(* CODESYS project FCC-Demo
   Author: Luke
   Company: Electra
   CompiledLibraryCompatibilityVersion: CODESYS V3.5 SP13
   Description: Reduced Brusa Temps for fan
      ePTO set to activate with reverse
      Cooling Fan reinstated
      Additional compressor run signals
      Gear change adjustment
      Comp temp Error SP raised
      Auto regen on overspeed >56@5s
      OR t AND for Traction Off Keypad Combo
   Title: e-Compact
   Version: 3.0.6

Project tree, tasks and I/O mapping:
  application Application
    libraries: SAE J1939, 3.0.9.1 (Epec Oy); Event Log, 3.3.0.0 (Epec Oy); CmpApp, * (System); CmpErrors, * (System); AD Conversion, 3.0.2.5 (Epec Oy); Analog Input, 3.0.0.5 (Epec Oy); CANopen, 3.5.4.3 (Epec Oy); CANopen 302, 3.0.2.2 (Epec Oy); CANopenCSDO, 3.1.3.1 (Epec Oy); CANopen OD Save, 3.3.3.8 (Epec Oy); Digital Output Diagnostic, 3.0.2.1 (Epec Oy); Event Log GUI, 3.0.1.9 (Epec Oy); Event Log Transfer, 3.0.4.4 (Epec Oy); RAM File System, 3.2.0.3 (Epec Oy); J1939 To Event Translator, 3.0.1.0 (Epec Oy); Filters, 3.0.1.4 (Epec Oy); Network Manager, 3.2.4.8 (Epec Oy); 5000types, 3.5.7.2 (Epec Oy); Joystick Calibration And Diagnostic, 3.2.0.6 (Epec Oy); Proportional Valve Control, 3.0.3.0 (Epec Oy); Ramp, 3.0.1.0 (Epec Oy); Sensor Calibration And Diagnostic, 3.0.1.6 (Epec Oy); DataTransfer, 3.0.2.0 (Epec Oy); CANVXD API, 4.0.0.1 (Epec Oy); Parameter Handler, 1.0.0.10 (Epec Oy); CANL2 CANVXD, 4.0.0.2 (Epec Oy); CANVXD API, 4.0.0.1 (Epec Oy); Util, * (System); BASIC, 3.3.4.0 (OSCAT)
    task PLC_PRG_TASK (cyclic, interval 10 ms, priority 1) calls PLC_PRG
    global variables ChangeLog
    CodeTemplate/
      Constants/
        global variables Code_Template_constants
      Enums/
        data type InitCanProtocolStates
      Globals/
        CANopen_CAN1/
          global variables G_CAN1_VAR
          global variables G_CANopen_CAN1
          global variables G_CANopen_CAN1_VAR
        CANopen_CAN2/
          global variables G_CAN2_VAR
          global variables G_CANopen_CAN2
          global variables G_CANopen_CAN2_VAR
        CANopen_CAN3/
          global variables G_CAN3_VAR
          global variables G_CANopen_CAN3
          global variables G_CANopen_CAN3_VAR
        CANopen_CAN4/
          global variables G_CAN4_VAR
          global variables G_CANopen_CAN4
          global variables G_CANopen_CAN4_VAR
        global variables Code_Template_globals
        global variables ERRORS
        global variables G_Common
        global variables G_SystemInfo
        global variables IO
        global variables IO_CONFIG
        global variables IO_INTERNAL
        global variables IO_RAW
        global variables J1939Globals
        global variables OD1_VAR
        global variables OD2_VAR
        global variables OD3_VAR
        global variables OD4_VAR
        global variables Slave_Configurations
        global variables SYSTEM
      POUs/
        program PLC_PRG [SFC]: Application_Action, Bus_Action, Diag_Action, EPEC_In_Action, Epec_Out_Action, Init_Action, Init_Bus_Action, Init_Entry_Action, Init_Events_Action, Init_Exit_Action, Init_Flash_Action, Init_IO_Action, Init_Protocols_Can1_Action, Init_Protocols_Can2_Action, Init_Protocols_Can3_Action, Init_Protocols_Can4_Action, IOFilter_Action, IOHandleOutputs_Action, Main_Application_Action, Other_Action, Other_EpecOut_Action
      Structs/
        CANopen/
          data type IdentityObject
        J1939/
          data type J1939_CAN1
          data type J1939_CAN1_IN
          data type J1939_CAN1_IN_BodyCont
          data type J1939_CAN1_IN_CCVS
          data type J1939_CAN1_IN_Engine
          data type J1939_CAN4
          data type J1939_CAN4_IN_ABS1
          data type J1939_CAN4_IN
          data type J1939_CAN4_IN_Tacho
    UserCode/
      BELDCDC/
        program BELDCDC_Control_1 [ST]
        program BELDCDC_Rx_1 [ST]
        program BELDCDC_RxConversion_1 [ST]
        program BELDCDC_Tx_1 [ST]
        program BELDCDC_TxConversion_1 [ST]
      BELDCDC/
        program BELDCDC_RxConversion [ST]
        program BELDCDC_Tx [ST]
        program BELDCDC_Control [ST]
        program BELDCDC_Rx [ST]
        program BELDCDC_TxConversion [ST]
        global variables BELDCDC_VAR
      BMS/
        global variables BMS_VAR
        program BMSData [ST]
        CATL/
          program CATLBMS_RxConversion [ST]
          program CATLBMS1_Rx [ST]
          global variables CATLBMS_VAR
        OrionBMS/
          program OrionBMS2_RxConversion [ST]
          global variables OrionBMS2_VAR
          program OrionBMS_Tx [ST]
          program Orion_Control [ST]
          program OrionBMS1_Rx [ST]
          program OrionBMS1_RxConversion [ST]
          global variables OrionBMS1_VAR
          program OrionBMS2_Rx [ST]
      BMS/
        global variables BMS_VAR_1
        program BMSData_1 [ST]
        CATL/
          program CATLBMS1_Rx_1 [ST]
          program CATLBMS_RxConversion_1 [ST]
          global variables CATLBMS_VAR_1
        OrionBMS/
          program Orion_Control_1 [ST]
          program OrionBMS1_Rx_1 [ST]
          program OrionBMS1_RxConversion_1 [ST]
          global variables OrionBMS1_VAR_1
          program OrionBMS2_Rx_1 [ST]
          program OrionBMS2_RxConversion_1 [ST]
          global variables OrionBMS2_VAR_1
          program OrionBMS_Tx_1 [ST]
      Brusa/
        Brusa1_Comms/
          program Brusa1_Rx_1 [ST]
          program Brusa1_RxConversion_1 [ST]
          program Brusa1_Tx_1 [ST]
          program Brusa1_TxConversion_1 [ST]
        Brusa2_Comms/
          program Brusa2_Rx_1 [ST]
          program Brusa2_RxConversion_1 [ST]
          program Brusa2_Tx_1 [ST]
          program Brusa2_TxConversion_1 [ST]
        program Brusa_1 [ST]: FreeContactor
        function block BrusaControl_1 [ST]: OkToCharge, OkToReset
      Brusa/
        Brusa1_Comms/
          program Brusa1_Rx [ST]
          program Brusa1_RxConversion [ST]
          program Brusa1_Tx [ST]
          program Brusa1_TxConversion [ST]
        Brusa2_Comms/
          program Brusa2_Rx [ST]
          program Brusa2_RxConversion [ST]
          program Brusa2_Tx [ST]
          program Brusa2_TxConversion [ST]
        program Brusa [ST]: FreeContactor
        function block BrusaControl [ST]: OkToCharge, OkToReset
      CAN1/
        program CAN1_RxConversion [ST]
        program CAN1_Rx [ST]
        program CAN1_TCMs_Tx [ST]
        program CAN1_Tx [ST]
        program CAN1_TxConversion [ST]
        global variables CAN1_VAR
        program KB_Tx [ST]
      CAN1/
        program CAN1_Rx_1 [ST]
        program CAN1_RxConversion_1 [ST]
        program CAN1_TCMs_Tx_1 [ST]
        program CAN1_Tx_1 [ST]
        program CAN1_TxConversion_1 [ST]
        global variables CAN1_VAR_1
        program KB_Tx_1 [ST]
      CAN3/
        program CAN3_Rx_1 [ST]
        program CAN3_RxConversion_1 [ST]
        program CAN3_Tx_1 [ST]
        global variables CAN3_VAR_1
      CAN3/
        program CAN3_RxConversion [ST]
        program CAN3_Rx [ST]
        program CAN3_Tx [ST]
        global variables CAN3_VAR
      CAN4/
        program CAN4_Rx [ST]
        program CAN4_Tx [ST]
        global variables CAN4_VAR
        global variables HMI_VAR
        program CAN4_TxConversion [ST]
        Data to or For HMI/
          program MCU_to_HMI [ST]
          program Sevcon_to_HMI [ST]
          program BMS_to_HMI [ST]
          program BRUSA_to_HMI [ST]
          program DCDC_to_HMI [ST]
          program VMU_to_HMI [ST]
        Heater/
          program Heater_Control [ST]
          global variables Heater_VAR
          program Heater_Rx [ST]
          program Heater_Tx [ST]
        program HMI_Rx [ST]
      CAN4/
        program CAN4_Rx_1 [ST]
        program CAN4_Tx_1 [ST]
        program CAN4_TxConversion_1 [ST]
        global variables CAN4_VAR_1
      CAN Function Blocks/
        CAN1/
          function block Receive_CAN1_EXD [ST]
          function block Callback_Receive_CAN1 [ST]: Receive
          function block Receive_CAN1_EXD_28bit [ST]
          function block Receive_CAN1_STD [ST]
        CAN3/
          function block Receive_CAN3_EXD_28bit [ST]
          function block Receive_CAN3_EXD [ST]
          function block Callback_Receive_CAN3 [ST]: Receive
          function block Receive_CAN3_STD [ST]
        data type t_CANReceive
        CAN2/
          function block Callback_Receive_CAN2 [ST]: Receive
          function block Receive_CAN2_EXD [ST]
          function block Receive_CAN2_STD [ST]
        CAN4/
          function block Receive_CAN4_EXD [ST]
          function block Callback_Receive_CAN4 [ST]: Receive
          function block Receive_CAN4_STD [ST]
      CAN Function Blocks/
        CAN1/
          function block Callback_Receive_CAN1_1 [ST]: Receive
          function block Receive_CAN1_EXD_1 [ST]
          function block Receive_CAN1_EXD_28bit_1 [ST]
          function block Receive_CAN1_STD_1 [ST]
        CAN2/
          function block Callback_Receive_CAN2_1 [ST]: Receive
          function block Receive_CAN2_EXD_1 [ST]
          function block Receive_CAN2_STD_1 [ST]
        CAN3/
          function block Callback_Receive_CAN3_1 [ST]: Receive
          function block Receive_CAN3_EXD_1 [ST]
          function block Receive_CAN3_EXD_28bit_1 [ST]
          function block Receive_CAN3_STD_1 [ST]
        CAN4/
          function block Callback_Receive_CAN4_1 [ST]: Receive
          function block Receive_CAN4_EXD_1 [ST]
          function block Receive_CAN4_STD_1 [ST]
        data type t_CANReceive_1
      CodeTemplateHandlers/
      Contactor Control/
        program ContactorControl_1 [ST]
      Contactor Control/
        program ContactorControl [ST]
      Cooling Fan/
        program Cooling_Fan [FBD]
      Cooling Fan/
        program Fan_Cooling [ST]
      Cruise Control/
        program CruiseControl [ST]
      DataTypes/
        data type tUpdate_1
      DataTypes/
        data type tUpdate
      ePTO/
        program EPTO_Rx [ST]
        global variables ePTO_VAR
        program ePTO_Control [ST]
        program EPTO_Tx [ST]
      ePTO/
        program ePTO_Control_1 [ST]
        program EPTO_Rx_1 [ST]
        program EPTO_Tx_1 [ST]
        global variables ePTO_VAR_1
      Fault Handler/
        program FaultDetection_1 [ST]
      Fault Handler/
        global variables Fault_VAR
        program FaultDetection [ST]
      Functions/
        function Update [ST]
      Functions/
        function Update_1 [ST]
      Heater/
        program Heater_Control_1 [ST]
        program Heater_Rx_1 [ST]
        program Heater_Tx_1 [ST]
      HMI/
        Data to or For HMI/
          program BMS_to_HMI_1 [ST]
          program BRUSA_to_HMI_1 [ST]
          program DCDC_to_HMI_1 [ST]
          program MCU_to_HMI_1 [ST]
          program Sevcon_to_HMI_1 [ST]
          program VMU_to_HMI_1 [ST]
        program HMI_Rx_1 [ST]
      Main Program/
        program Chassis_Parameters [ST]
        program ComponentSelection [ST]
        program Main [ST]: IO_Reconfiguration
        global variables PersistentVars
        program System_StateSpace [ST]
        function GetAppInfo [ST]
        global variables Main_VAR
        program MainInit [ST]
        program Project_Infomation [FBD]
        program RealTimeClock [FBD]
      MCU/
        program Dennis_Regen [FBD]
        program Driveability [ST]
        function f_DistanceCalc [ST]
        function f_SpeedCalc [ST]
        program MCU_Control [ST]
        program MCU_Rx [ST]
        program GearSelection [ST]
        program MCU_RxConversion [ST]
        program MCU_Tx [ST]
        program MCU_TxConversion [ST]
        global variables MCU_VAR
      MCU/
        program Dennis_Regen_1 [FBD]
        program Driveability_1 [ST]
        function f_DistanceCalc_1 [ST]
        function f_SpeedCalc_1 [ST]
        program GearSelection_1 [ST]
        program MCU_Control_1 [ST]
        program MCU_Rx_1 [ST]
        program MCU_RxConversion_1 [ST]
        program MCU_Tx_1 [ST]
        program MCU_TxConversion_1 [ST]
        global variables MCU_VAR_1
      Sevcon_Compressor/
        program Sevcon2_Rx [ST]
        program Sevcon2_RxConversion [ST]
        program Sevcon2_TxConversion [ST]
        global variables Sevcon2_VAR
        program Sevcon2_Control [ST]
        program Sevcon2_Tx [ST]
      Sevcon_Compressor/
        program Sevcon2_Control_1 [ST]
        program Sevcon2_Rx_1 [ST]
        program Sevcon2_RxConversion_1 [ST]
        program Sevcon2_Tx_1 [ST]
        program Sevcon2_TxConversion_1 [ST]
        global variables Sevcon2_VAR_1
      Sevcon ePTO/
        program Sevcon_ePTO_Control [ST]
        program Sevcon_ePTO_Rx [ST]
        program Sevcon_ePTO_RxConversion [ST]
        program Sevcon_ePTO_Tx [ST]
        program Sevcon_ePTO_TxConversion [ST]
        global variables Sevcon_ePTO_VAR
      Sevcon_PSP/
        program Sevcon_Steer_Control [ST]
        program Sevcon_Steer_Rx [ST]
        program Sevcon_Steer_RxConversion [ST]
        program Sevcon_Steer_Tx [ST]
        program Sevcon_Steer_TxConversion [ST]
        global variables Sevcon_Steer_VAR
      Sevcon_PSP/
        program Sevcon_Steer_Control_1 [ST]
        program Sevcon_Steer_Rx_1 [ST]
        program Sevcon_Steer_RxConversion_1 [ST]
        program Sevcon_Steer_Tx_1 [ST]
        program Sevcon_Steer_TxConversion_1 [ST]
        global variables Sevcon_Steer_VAR_1
      UserMramUsage_1/
        data type UserMRAMStructure_1
        global variables UserMramVariables_1
      UserMramUsage/
        data type UserMRAMStructure
        global variables UserMramVariables
  function GetLibVersion [ST]
  function GetLibVersionNumber [ST]
  function IsLibReleased [ST]
  function GetBooleanProperty [ST]
  function GetCompany [ST]
  function GetNumberProperty [ST]
  function GetTextProperty2 [ST]
  function GetTextProperty [ST]
  function GetTitle [ST]
  function GetVersion [ST]
  function GetVersionProperty [ST]
*)

// Application/CodeTemplate/Enums/InitCanProtocolStates
TYPE InitCanProtocolStates :
(
	INIT_CANOPEN_PROTOCOLS := 1,
	INIT_CANOPEN_OD := 2,
	INIT_CANOPEN_PDO := 3,
	INIT_CANOPEN_OD_SAVE := 4,
	INIT_J1939 := 5,
	INIT_PROTOCOLS_DONE := 6
);
END_TYPE

// Application/UserCode/CAN Function Blocks/t_CANReceive
TYPE t_CANReceive EXTENDS EPEC_CANL2.EPEC_CANVXD.Msg:
STRUCT
	q_NewDataRxed	:	BOOL;
END_STRUCT
END_TYPE

// Application/UserCode/CAN Function Blocks/t_CANReceive_1
TYPE t_CANReceive_1 EXTENDS EPEC_CANL2.EPEC_CANVXD.Msg:
STRUCT
	q_NewDataRxed	:	BOOL;
END_STRUCT
END_TYPE

// Application/UserCode/DataTypes/tUpdate_1
(*================================================================================================*)
(*   Screen Update Structure                                                                      *)
(*================================================================================================*)
 TYPE tUpdate_1 :
 STRUCT
  Step	        :BYTE  := 0;   // Current State
  Next	        :BYTE  := 0;   // Requested Next State 
  Last	        :BYTE  := 0;   // Last Active State
  Force	        :BYTE  := 255; // Forced Next State	
  Tmr		    :WORD  := 0;   // Time In State
  Seq		    :DWORD := 0;   // Last 4 States 

 END_STRUCT
 END_TYPE

// Application/UserCode/UserMramUsage_1/UserMRAMStructure_1
TYPE UserMRAMStructure_1 :
STRUCT
   (* Header part *)
    UserMRAMdataValid:BOOL := FALSE;	(* 	Set TRUE if data pointer is initialised correctly else set FALSE*) 
    UserMRAMinitError:INT := 0; 		(* 	Possible errors 
                    						0 = SUCCESS, 
											1 = Structure size is too big to fit in MRAM, 
											2 = Tag not AA55AA55h *)                                                         
    UserMRAMTag:DWORD:=16#AA55AA55; 	(* Tag value must always be AA55AA55h *)

	(* 	User part. Forward from here user can add own variables which are stored in MRAM.
    	NOTE!!! You can add structure members until structure size is bigger than reserved size.
        In of error in size of the MRAM pointer from system pointer G_pUserMramStructure is set to point default instance
        G_UserMramStructureDefault and dataValid is set FALSE.

        NOTE!!! It is allowed to add pointers to end of the structure but not in the between 
        already added structure members.*)

		
		
END_STRUCT
END_TYPE

// Application/UserCode/UserMramUsage/UserMRAMStructure
TYPE UserMRAMStructure :
STRUCT
   (* Header part *)
    UserMRAMdataValid:BOOL := FALSE;	(* 	Set TRUE if data pointer is initialised correctly else set FALSE*) 
    UserMRAMinitError:INT := 0; 		(* 	Possible errors 
                    						0 = SUCCESS, 
											1 = Structure size is too big to fit in MRAM, 
											2 = Tag not AA55AA55h *)                                                         
    UserMRAMTag:DWORD:=16#AA55AA55; 	(* Tag value must always be AA55AA55h *)

	(* 	User part. Forward from here user can add own variables which are stored in MRAM.
    	NOTE!!! You can add structure members until structure size is bigger than reserved size.
        In of error in size of the MRAM pointer from system pointer G_pUserMramStructure is set to point default instance
        G_UserMramStructureDefault and dataValid is set FALSE.

        NOTE!!! It is allowed to add pointers to end of the structure but not in the between 
        already added structure members.*)

		
		
END_STRUCT
END_TYPE

// Application/CodeTemplate/Structs/CANopen/IdentityObject
TYPE IdentityObject :
STRUCT
	///Vendor ID
	VendorId: DWORD := 0;
	///Product code
	ProductCode: DWORD := 0;
	///Revision number
	Revision: DWORD := 0;
	///Serial number for control unit
	SerialNumber: DWORD := 0;
END_STRUCT
END_TYPE

// Application/CodeTemplate/Structs/J1939/J1939_CAN1
TYPE J1939_CAN1 :
STRUCT
	In: J1939_CAN1_IN;
END_STRUCT
END_TYPE

// Application/CodeTemplate/Structs/J1939/J1939_CAN1_IN
TYPE J1939_CAN1_IN :
STRUCT
	BodyCont: J1939_CAN1_IN_BodyCont;
	Engine: J1939_CAN1_IN_Engine;
	CCVS: J1939_CAN1_IN_CCVS;
	PGNs: ARRAY[1..3] OF J1939_pPGN;
END_STRUCT
END_TYPE

// Application/CodeTemplate/Structs/J1939/J1939_CAN1_IN_BodyCont
TYPE J1939_CAN1_IN_BodyCont :
STRUCT
	AIR1_PneumaticSupplyPress: BYTE;
	AIR1_ParkingAnd_OrTrailerAirPress: BYTE;
	AIR1_ServiceBrakeAirPressCircuit1: BYTE;
	AIR1_ServiceBrakeAirPressCircuit2: BYTE;
	AIR1_AuxEquipmentSupplyPress: BYTE;
	AIR1_AirSuspensionSupplyPress: BYTE;
	AIR1_AirCompressorStatus: BYTE;
	PGN_AIR1_SPNs: ARRAY[1..7] OF J1939_SPN;
	PGN_AIR1: J1939_PGN;
END_STRUCT
END_TYPE

// Application/CodeTemplate/Structs/J1939/J1939_CAN1_IN_CCVS
TYPE J1939_CAN1_IN_CCVS :
STRUCT
	CCVS_TwoSpeedAxleSwitch: BYTE;
	CCVS_ParkingBrakeSwitch: BYTE;
	CCVS_CruiseCtrlPauseSwitch: BYTE;
	CCVS_ParkBrakeReleaseInhibitRq: BYTE;
	CCVS_WheelBasedVehicleSpeed: WORD;
	CCVS_CruiseCtrlActive: BYTE;
	CCVS_CruiseCtrlEnableSwitch: BYTE;
	CCVS_BrakeSwitch: BYTE;
	CCVS_ClutchSwitch: BYTE;
	CCVS_CruiseCtrlSetSwitch: BYTE;
	CCVS_CruiseCtrlCoastSwitch: BYTE;
	CCVS_CruiseCtrlResumeSwitch: BYTE;
	CCVS_CruiseCtrlAccelerateSwitch: BYTE;
	CCVS_CruiseCtrlSetSpeed: BYTE;
	CCVS_PTOState: BYTE;
	CCVS_CruiseCtrlStates: BYTE;
	CCVS_EngIdleIncrementSwitch: BYTE;
	CCVS_EngIdleDecrementSwitch: BYTE;
	CCVS_EngTestModeSwitch: BYTE;
	CCVS_EngShutdownOverrideSwitch: BYTE;
	PGN_CCVS_SPNs: ARRAY[1..20] OF J1939_SPN;
	PGN_CCVS: J1939_PGN;
END_STRUCT
END_TYPE

// Application/CodeTemplate/Structs/J1939/J1939_CAN1_IN_Engine
TYPE J1939_CAN1_IN_Engine :
STRUCT
	EEC2_AccelPedal1LowIdleSwitch: BYTE;
	EEC2_AccelPedalKickdownSwitch: BYTE;
	EEC2_RoadSpeedLimitStatus: BYTE;
	EEC2_AccelPedal2LowIdleSwitch: BYTE;
	EEC2_AccelPedalPos1: BYTE;
	EEC2_EngPercentLoadAtCurrentSpeed: BYTE;
	EEC2_RemoteAccelPedalPos: BYTE;
	EEC2_AccelPedalPos2: BYTE;
	EEC2_VhclAccelerationRateLimitStatus: BYTE;
	J1939_CAN1_EEC2_Dummy_RX_1: BYTE;
	EEC2_ActMaxAvailEngPercentTorque: BYTE;
	PGN_EEC2_SPNs: ARRAY[1..11] OF J1939_SPN;
	PGN_EEC2: J1939_PGN;
END_STRUCT
END_TYPE

// Application/CodeTemplate/Structs/J1939/J1939_CAN4
TYPE J1939_CAN4 :
STRUCT
	In: J1939_CAN4_IN;
END_STRUCT
END_TYPE

// Application/CodeTemplate/Structs/J1939/J1939_CAN4_IN_ABS1
TYPE J1939_CAN4_IN_ABS1 :
STRUCT
	EBC1_ASREngCtrlActive: BYTE;
	EBC1_ASRBrakeCtrlActive: BYTE;
	EBC1_AntiLockBrakingActive: BYTE;
	EBC1_EBSBrakeSwitch: BYTE;
	EBC1_BrakePedalPos: BYTE;
	EBC1_ABSOffroadSwitch: BYTE;
	EBC1_ASROffroadSwitch: BYTE;
	EBC1_ASRHillHolderSwitch: BYTE;
	EBC1_TractionCtrlOverrideSwitch: BYTE;
	EBC1_AccelInterlockSwitch: BYTE;
	EBC1_EngDerateSwitch: BYTE;
	EBC1_EngAuxEngShutdownSwitch: BYTE;
	EBC1_RemoteAccelEnableSwitch: BYTE;
	EBC1_EngRetarderSelection: BYTE;
	EBC1_ABSFullyOperational: BYTE;
	EBC1_EBSRedWarningSignal: BYTE;
	EBC1_ABS_EBSAmberWarningSignal: BYTE;
	EBC1_ATC_ASRInformationSignal: BYTE;
	EBC1_SrcAddrssOfCtrllngDvcFrBrkCntrl: BYTE;
	J1939_CAN4_EBC1_Dummy_RX_1: BYTE;
	EBC1_HaltBrakeSwitch: BYTE;
	EBC1_TrailerABSStatus: BYTE;
	EBC1_TrctrMntdTrilerABSWarningSignal: BYTE;
	PGN_EBC1_SPNs: ARRAY[1..23] OF J1939_SPN;
	PGN_EBC1: J1939_PGN;
END_STRUCT
END_TYPE

// Application/CodeTemplate/Structs/J1939/J1939_CAN4_IN
TYPE J1939_CAN4_IN :
STRUCT
	ABS1: J1939_CAN4_IN_ABS1;
	Tacho: J1939_CAN4_IN_Tacho;
	PGNs: ARRAY[1..3] OF J1939_pPGN;
END_STRUCT
END_TYPE

// Application/CodeTemplate/Structs/J1939/J1939_CAN4_IN_Tacho
TYPE J1939_CAN4_IN_Tacho :
STRUCT
	TD_Seconds: BYTE;
	TD_Minutes: BYTE;
	TD_Hours: BYTE;
	TD_Month: BYTE;
	TD_Day: BYTE;
	TD_Year: BYTE;
	TD_LocalMinuteOffset: BYTE;
	TD_LocalHourOffset: BYTE;
	PGN_TD_SPNs: ARRAY[1..8] OF J1939_SPN;
	PGN_TD: J1939_PGN;
	VD_TripDistance: DWORD;
	VD_TotalVehicleDistance: DWORD;
	PGN_VD_SPNs: ARRAY[1..2] OF J1939_SPN;
	PGN_VD: J1939_PGN;
END_STRUCT
END_TYPE

// Application/UserCode/DataTypes/tUpdate
(*================================================================================================*)
(*   Screen Update Structure                                                                      *)
(*================================================================================================*)
 TYPE tUpdate :
 STRUCT
  Step	        :BYTE  := 0;   // Current State
  Next	        :BYTE  := 0;   // Requested Next State 
  Last	        :BYTE  := 0;   // Last Active State
  Force	        :BYTE  := 255; // Forced Next State	
  Tmr		    :WORD  := 0;   // Time In State
  Seq		    :DWORD := 0;   // Last 4 States 

 END_STRUCT
 END_TYPE

// Application/ChangeLog
{attribute 'qualified_only'}
VAR_GLOBAL
(*
TEST Version H
Motor Temp 100-120
Cut in pressure 8bar
Full Regen on Brake
Set regenValue to MAX on startup
Variables for PSP instead of constants
Reduced PSP speed instead of OFF
Steering active on handbrake OFF OR <>Neutral


*)	


END_VAR

// Application/CodeTemplate/Constants/Code_Template_constants
VAR_GLOBAL CONSTANT
	///Size for the area which is used for parameter system. This area is reserved from the beginning of the MRAM area which is reserved for usage for PLCopn application. 
	G_MRAM_AREA_SIZE_FOR_PAR_SYS: DWORD := 16#19000;
	///Number of parameters in network
	G_NUMBER_OF_PARAMETERS_NETWORK1: INT := 0;
	///Number of parameters in network
	G_NUMBER_OF_PARAMETERS_NETWORK2: INT := 0;
	///Number of parameters in network
	G_NUMBER_OF_PARAMETERS_NETWORK3: INT := 0;
	///Number of parameters in network
	G_NUMBER_OF_PARAMETERS_NETWORK4: INT := 0;
	/// Parameterhandler keyword
	G_PARAMHANDLERKEYWORD: DWORD := 16#4F792812;
	/// Maximum size of one parameter handler block
	G_PARAM_BLOCK_MAX_SIZE: WORD := 1024;
END_VAR

// Application/CodeTemplate/Globals/Code_Template_globals
VAR_GLOBAL
	///Function block for HWD_Measurements.
	G_HWDiagnostics: HWD_Measurements;
	///Flag indicates if unit is wanted to reset after current application cycle. Reset actions can be varied between platforms.
	G_RESET_MODULE: BOOL := FALSE;
	///Add all automatically generated events to log.
	G_AddAllAutoGenEventsToLog: BOOL := TRUE;
	///Off delay for automatically generated events.
	G_OffDelayForAutoGenEvents: WORD := 50;
	///On delay for automatically generated events.
	G_OnDelayForAutoGenEvents: WORD := 0;
	///Variable defines low limit for parameter saving [0.01V]. Compared votlage is read from HWD_Measurements function block. If read voltage is smaller than defined value parameter saving is not started.
	G_LowLimitForParameterSaving: WORD := 900;
	///Pin 1.9 - Function block instance for AI protection.
	G_AIprotection_X1_09: AI_INPUTPROTECTION;
	///Pin 1.10 - Function block instance for AI protection.
	G_AIprotection_X1_10: AI_INPUTPROTECTION;
	///Pin 1.11 - Function block instance for Debounce
	G_DebounceDI_q_BatteryInterlockIn_DI: Filters_DebounceDI_Fast;
	///Pin 1.20 - Function block instance for AI protection.
	G_AIprotection_X1_20: AI_INPUTPROTECTION;
	///Pin 1.21 - Function block instance for AI protection.
	G_AIprotection_X1_21: AI_INPUTPROTECTION;
	///Pin 2.6 - Function block instance for Debounce
	G_DebounceDI_q_Battery1ChargeRq_DI: Filters_DebounceDI_Fast;
	///Pin 2.7 - Function block instance for Debounce
	G_DebounceDI_q_Battery1DiscahrgeRq_DI: Filters_DebounceDI_Fast;
	///Pin 2.8 - Function block instance for Debounce
	G_DebounceDI_q_Battery2ChargeRq_DI: Filters_DebounceDI_Fast;
	///Pin 2.9 - Function block instance for Debounce
	G_DebounceDI_q_Batter2DischargeRq_DI: Filters_DebounceDI_Fast;
	///Pin 2.16 - Function block instance for Debounce
	G_DebounceDI_q_ChargePlugLockStatus_DI: Filters_DebounceDI_Fast;
	///Pin 2.23 - Function block instance for AI protection.
	G_AIprotection_X2_23: AI_INPUTPROTECTION;
	///Pin 3.5 - Function block instance for Debounce
	G_DebounceDI_q_DirectionSwitch_ReverseCrawl_DI: Filters_DebounceDI_Fast;
	///Pin 3.6 - Function block instance for Debounce
	G_DebounceDI_q_DirectionSwitch_Drive_DI: Filters_DebounceDI_Fast;
	///Pin 3.7 - Function block instance for Debounce
	G_DebounceDI_q_IlluminiationStatsus_DI: Filters_DebounceDI_Fast;
	///Pin 3.8 - Function block instance for Debounce
	G_DebounceDI_q_DirectionSwitch_Reverse_DI: Filters_DebounceDI_Fast;
	///Pin 3.9 - Function block instance for Debounce
	G_DebounceDI_q_DirectionSwitch_DriveCrawl_DI: Filters_DebounceDI_Fast;
	///Pin 3.11 - Function block instance for Debounce
	G_DebounceDI_q_DirectionSwitch_Neutral_DI: Filters_DebounceDI_Fast;
	///Pin 3.12 - Function block instance for Debounce
	G_DebounceDI_q_DoorOpen_DI: Filters_DebounceDI_Fast;
	///Pin 3.14 - Function block instance for AI protection.
	G_AIprotection_X3_14: AI_INPUTPROTECTION;
	///Pin 3.15 - Function block instance for AI protection.
	G_AIprotection_X3_15: AI_INPUTPROTECTION;
	///Pin 3.16 - Function block instance for AI protection.
	G_AIprotection_X3_16: AI_INPUTPROTECTION;
	///Pin 3.22 - Function block instance for Debounce
	G_DebounceDI_q_VehicleKL15_DI: Filters_DebounceDI_Fast;
	///Pin 3.23 - Function block instance for Debounce
	G_DebounceDI_q_VehicleKL51_DI: Filters_DebounceDI_Fast;
	///Pin 3.28 - Function block instance for Debounce
	G_DebounceDI_q_HeaterIn_DI: Filters_DebounceDI_Fast;
	G_SystemOk: BOOL := FALSE;
	G_TempHighLimit: INT := 1050;
	G_TempLowLimit: INT := -400;
	G_SupplyVoltageHighLimit: INT := 3000;
	G_SupplyVoltageLowLimit: INT := 1400;
	G_CycleTimeHighLimit: INT := 30;
	G_Ref5VHighLimit: INT := 550;
	G_Ref5VLowLimit: INT := 450;
	G_Ref10VHighLimit: INT := 1050;
	G_Ref10VLowLimit: INT := 950;
	G_PullUp10VHighLimit: INT := 1050;
	G_PullUp10VLowLimit: INT := 950;
	G_RefADCVHighLimit: INT := 150;
	G_RefADCVLowLimit: INT := 100;
	///Init Flags
	G_InitEntryReady: BOOL := FALSE;
	G_InitFlashReady: BOOL := FALSE;
	G_InitIOReady: BOOL := FALSE;
	G_InitBusReady: BOOL := FALSE;
	G_InitProtocolsCan1Ready: BOOL := FALSE;
	G_InitProtocolsCan2Ready: BOOL := FALSE;
	G_InitProtocolsCan3Ready: BOOL := FALSE;
	G_InitProtocolsCan4Ready: BOOL := FALSE;
	G_InitEventsReady: BOOL := FALSE;
	G_InitExitReady: BOOL := FALSE;
	G_ActiveError: BOOL := FALSE;
	///Global variable which is used to store result value from POU calls.
	G_ShmUserMRAM: SysSharedMemRegion;
	///Global variable which is used to store result value from POU calls.
	G_FunctionResult: CmpApp.RTS_IEC_RESULT;
	///Global variable which is used to store result value from POU calls.
	G_MramStartAddressForUser: DWORD;
	///Global variable which is used to store result value from POU calls.
	G_MramEndAddressForUser: DWORD;
	G_MramInitErrors: INT := 0;
	G_CounterRestoreCmdOld: WORD := 0;
	G_CounterSaveCmdOld: WORD := 0;
	G_NodeIds: ARRAY[1..4] OF INT := [1, 1, 1, 1];
	G_CAN1_Channel: EPEC_CANL2.Channel;
	G_InitProtocolsCan1State: InitCanProtocolStates := INIT_CANOPEN_PROTOCOLS;
	G_InitCANopenCan1Error: BOOL := FALSE;
	G_CANopenCan1ProtocolError: BOOL := FALSE;
	G_CAN2_Channel: EPEC_CANL2.Channel;
	G_InitProtocolsCan2State: InitCanProtocolStates := INIT_CANOPEN_PROTOCOLS;
	G_InitCANopenCan2Error: BOOL := FALSE;
	G_CANopenCan2ProtocolError: BOOL := FALSE;
	G_CAN3_Channel: EPEC_CANL2.Channel;
	G_InitProtocolsCan3State: InitCanProtocolStates := INIT_CANOPEN_PROTOCOLS;
	G_InitCANopenCan3Error: BOOL := FALSE;
	G_CANopenCan3ProtocolError: BOOL := FALSE;
	G_CAN4_Channel: EPEC_CANL2.Channel;
	G_InitProtocolsCan4State: InitCanProtocolStates := INIT_CANOPEN_PROTOCOLS;
	G_InitCANopenCan4Error: BOOL := FALSE;
	G_CANopenCan4ProtocolError: BOOL := FALSE;
END_VAR

// Application/CodeTemplate/Globals/ERRORS
VAR_GLOBAL
	///Flag is set true if there is at least one monitored error in I/O init functions.
	ERR_FLAG_IO_INIT: BOOL := FALSE;
	///Pin 1.9 - Error flag is raised if over current is occured for AI pin which is used in mA mode.
	ERR_FLAG_IO_AI_OVER_CURRENT_X1_09: BOOL := FALSE;
	///Pin 1.10 - Error flag is raised if over current is occured for AI pin which is used in mA mode.
	ERR_FLAG_IO_AI_OVER_CURRENT_X1_10: BOOL := FALSE;
	///Pin 1.20 - Error flag is raised if over current is occured for AI pin which is used in mA mode.
	ERR_FLAG_IO_AI_OVER_CURRENT_X1_20: BOOL := FALSE;
	///Pin 1.21 - Error flag is raised if over current is occured for AI pin which is used in mA mode.
	ERR_FLAG_IO_AI_OVER_CURRENT_X1_21: BOOL := FALSE;
	///Pin 2.23 - Error flag is raised if over current is occured for AI pin which is used in mA mode.
	ERR_FLAG_IO_AI_OVER_CURRENT_X2_23: BOOL := FALSE;
	///Pin 3.14 - Error flag is raised if over current is occured for AI pin which is used in mA mode.
	ERR_FLAG_IO_AI_OVER_CURRENT_X3_14: BOOL := FALSE;
	///Pin 3.15 - Error flag is raised if over current is occured for AI pin which is used in mA mode.
	ERR_FLAG_IO_AI_OVER_CURRENT_X3_15: BOOL := FALSE;
	///Pin 3.16 - Error flag is raised if over current is occured for AI pin which is used in mA mode.
	ERR_FLAG_IO_AI_OVER_CURRENT_X3_16: BOOL := FALSE;
END_VAR

// Application/CodeTemplate/Globals/G_Common
{attribute 'qualified_only' := ''}
VAR_GLOBAL
	///Parameterhandler. Utility library for ODSave. Library handles parameter image modification. 
	ParHandler: EPEC_PH.ParameterHandler;
	/// Project key, used for validating the response code
	ProjectKey: STRING(79) := '3J0YxHBXH5eQbnz';
END_VAR

// Application/CodeTemplate/Globals/G_SystemInfo
///
///            NOTE! NOTE! NOTE! NOTE! NOTE! NOTE! NOTE! NOTE! NOTE! NOTE! NOTE!
///
///            This object is created by Epec MultiTool.
///            User changes are overwritten when project is imported.
///
///            Content:
///            - System information common for all ODs.
///
///          
{attribute 'qualified_only' := ''}
VAR_GLOBAL
	ProjectInfo: CmpApp.PROJECT_INFO;
	/// 16#1008: Manufacturer device name
	DeviceName: STRING(79);
	/// 16#1009: Manufacturer hardware version
	HWVersion: STRING(79);
	/// 16#100A: Manufacturer software version
	SWVersion: STRING(79);
	/// 16#1018: Identity object 
	Identity: IdentityObject;
	/// 16#2030 Codesys version
	ToolsVersionInfo: ARRAY[1..1] OF DWORD := [DWORD#50659328];
	FWErrorLog: POINTER TO SysErrorLogData;
	/// 16#2130 Software information
	/// Sub1: Application version
	/// Sub2: Additional version information
	/// Sub3: Reserved for future use
	/// Sub4: Reserved for future use
	/// Sub5: Reserved for future use
	/// Sub6: Reserved for future use
	/// Sub7: Reserved for future use
	/// Sub8: Reserved for future use
	/// Sub9: Reserved for future use
	/// Sub10: Reserved for future use
	SoftwareInformation: ARRAY[1..10] OF STRING(79) := [''];
	/// 16#2140 MAC address
	/// Sub1: MAC address byte 1
	/// Sub2: MAC address byte 2
	/// Sub3: MAC address byte 3
	/// Sub4: MAC address byte 4
	/// Sub5: MAC address byte 5
	/// Sub6: MAC address byte 6
	MACAddress: ARRAY[1..6] OF BYTE := [6(0)];
	/// 16#2141 Ethernet configuration
	/// Sub1: Ethernet enabled/disabled
	/// Sub2: DHCP on/off
	/// Sub3: Reserved
	/// Sub4: Reserved
	/// Sub5: Reserved
	/// Sub6: Reserved
	/// Sub7: Reserved
	/// Sub8: Reserved
	/// Sub9: Reserved
	/// Sub10: Reserved
	/// Sub11: Reserved
	/// Sub12: Reserved
	/// Sub13: Reserved
	/// Sub14: Reserved
	/// Sub15: Reserved
	/// Sub16: Reserved
	/// Sub17: Reserved
	/// Sub18: Netstatus
	/// Sub19: IP address highest byte
	/// Sub20: IP address 3rd byte
	/// Sub21: IP address 2nd byte
	/// Sub22: IP address lowest byte
	/// Sub23: Gateway highest byte
	/// Sub24: Gateway 3rd byte
	/// Sub25: Gateway 2nd byte
	/// Sub26: Gateway lowest byte
	/// Sub27: Netmask highest byte
	/// Sub28: Netmask 3rd byte
	/// Sub29: Netmask 2nd byte
	/// Sub30: Netmask first byte
	/// Sub31: Reserved
	/// Sub32: Reserved
	/// Sub33: Reserved
	/// Sub34: Reserved
	/// Sub35: Reserved
	/// Sub36: Reserved
	/// Sub37: Reserved
	/// Sub38: Reserved
	/// Sub39: Reserved
	/// Sub40: Reserved
	/// Sub41: Reserved
	/// Sub42: Reserved
	/// Sub43: Reserved
	/// Sub44: Reserved
	/// Sub45: Reserved
	/// Sub46: Reserved
	/// Sub47: Reserved
	/// Sub48: Reserved
	/// Sub49: Reserved
	/// Sub50: Reserved
	EthernetConfiguration: ARRAY[1..50] OF BYTE := [50(0)];
	/// 16#2150 CAN 1 Communication parameters
	/// Sub1: CODESYS communication enabled
	/// Sub2: CODESYS communication node-ID
	/// Sub3: Bit rate
	/// Sub4: Cable detection offset for CODESYS node-ID
	/// Sub5: Cable detection offset for PLCopen node-ID
	/// Sub6: Mask for cable detection pins
	/// Sub7: Reserved
	/// Sub8: Reserved
	/// Sub9: Reserved
	/// Sub10: PLCopen application node-ID in CAN1
	CAN1_Comms: ARRAY[1..10] OF WORD := [10(0)];
	/// 16#2151 CAN 2 Communication parameters
	/// Sub1: CODESYS communication enabled
	/// Sub2: CODESYS communication node-ID
	/// Sub3: Bit rate
	/// Sub4: Reserved
	/// Sub5: Reserved
	/// Sub6: Reserved
	/// Sub7: Reserved
	/// Sub8: Reserved
	/// Sub9: Reserved
	/// Sub10: PLCopen application node-ID in CAN2
	CAN2_Comms: ARRAY[1..10] OF WORD := [10(0)];
	/// 16#2152 CAN 3 Communication parameters
	/// Sub1: CODESYS communication enabled
	/// Sub2: CODESYS communication node-ID
	/// Sub3: Bit rate
	/// Sub4: Reserved
	/// Sub5: Reserved
	/// Sub6: Reserved
	/// Sub7: Reserved
	/// Sub8: Reserved
	/// Sub9: Reserved
	/// Sub10: PLCopen application node-ID in CAN3
	CAN3_Comms: ARRAY[1..10] OF WORD := [10(0)];
	/// 16#2153 CAN 4 Communication parameters
	/// Sub1: CODESYS communication enabled
	/// Sub2: CODESYS communication node-ID
	/// Sub3: Bit rate
	/// Sub4: Reserved
	/// Sub5: Reserved
	/// Sub6: Reserved
	/// Sub7: Reserved
	/// Sub8: Reserved
	/// Sub9: Reserved
	/// Sub10: PLCopen application node-ID in CAN4
	CAN4_Comms: ARRAY[1..10] OF WORD := [10(0)];
END_VAR

// Application/CodeTemplate/Globals/IO
VAR_GLOBAL
	///Pin 1.9 - Filtered AI value
	AIPU_u16_DrivetrainTemp_AI: WORD := 0;
	///Pin 1.9 - Filtered AI value
	AI_u16_DrivetrainTemp_AI: WORD := 0;
	///Pin 1.10 - Filtered AI value
	AIPU_u16_ChargePlugPresent_AI: WORD := 0;
	///Pin 1.10 - Filtered AI value
	AI_u16_ChargePlugPresent_AI: WORD := 0;
	///Pin 1.11 - Filtered digital input status.
	DI_q_BatteryInterlockIn_DI: BOOL := FALSE;
	///Pin 1.12 - Digital output status for output pin.
	DO_q_BackupPump_DO AT %QX89.8: BOOL := FALSE;
	///Pin 1.12 - Current feedback for output [0..2500 mA].
	PWFM_CM_q_BackupPump_DO AT %IB132: DWORD := 0;
	///Pin 1.12 - Digital input state for pin.
	DOS_q_BackupPump_DO AT %IX768.8: BOOL := FALSE;
	///Pin 1.12 - State of the overcurrent error.
	PWFM_OVERCURRENT_q_BackupPump_DO AT %IX70.12: BOOL := FALSE;
	///Pin 1.12 - State of the broken circuit error. Demands firmware version 1.2.X to work correctly. Not supported for step motor mode. For firmware versions for which brokent circuit is supported current limit can be set with function IO_PWFM_SET_BRK_DIAG_CURRENT.
	PWFM_OPENCIRCUIT_q_BackupPump_DO AT %IX70.14: BOOL := FALSE;
	///Pin 1.20 - Filtered AI value
	AIPU_u16_Heater1Temperature_AI: WORD := 0;
	///Pin 1.20 - Filtered AI value
	AI_u16_Heater1Temperature_AI: WORD := 0;
	///Pin 1.21 - Filtered AI value
	AIPU_u16_Heater2Temperature_AI: WORD := 0;
	///Pin 1.21 - Filtered AI value
	AI_u16_Heater2Temperature_AI: WORD := 0;
	///Pin 1.22 - Digital output status for output pin.
	DO_q_BatteryDischargeMain_DO AT %QX209.8: BOOL := FALSE;
	///Pin 1.22 - Digital input state for pin.
	DOS_q_BatteryDischargeMain_DO AT %IX770.8: BOOL := FALSE;
	///Pin 1.23 - Digital output status for output pin.
	DO_q_AirPressureReliefValve_DO AT %QX99.8: BOOL := FALSE;
	///Pin 1.23 - Current feedback for output [0..2500 mA].
	PWFM_CM_q_AirPressureReliefValve_DO AT %IB148: DWORD := 0;
	///Pin 1.23 - Digital input state for pin.
	DOS_q_AirPressureReliefValve_DO AT %IX768.9: BOOL := FALSE;
	///Pin 1.23 - State of the overcurrent error.
	PWFM_OVERCURRENT_q_AirPressureReliefValve_DO AT %IX78.12: BOOL := FALSE;
	///Pin 1.23 - State of the broken circuit error. Demands firmware version 1.2.X to work correctly. Not supported for step motor mode. For firmware versions for which brokent circuit is supported current limit can be set with function IO_PWFM_SET_BRK_DIAG_CURRENT.
	PWFM_OPENCIRCUIT_q_AirPressureReliefValve_DO AT %IX78.14: BOOL := FALSE;
	///Pin 1.29 - Digital output status for output pin.
	DO_q_Battery1ChargePrecharge_DO AT %QX279.8: BOOL := FALSE;
	///Pin 1.29 - Digital input state for pin.
	DOS_q_Battery1ChargePrecharge_DO AT %IX770.15: BOOL := FALSE;
	///Pin 1.30 - Digital output status for output pin.
	DO_q_Battery1ChargeMain_DO AT %QX269.8: BOOL := FALSE;
	///Pin 1.30 - Digital input state for pin.
	DOS_q_Battery1ChargeMain_DO AT %IX770.14: BOOL := FALSE;
	///Pin 1.31 - Digital output status for output pin.
	DO_q_Battery2ChargePrecharge_DO AT %QX259.8: BOOL := FALSE;
	///Pin 1.31 - Digital input state for pin.
	DOS_q_Battery2ChargePrecharge_DO AT %IX770.13: BOOL := FALSE;
	///Pin 1.32 - Digital output status for output pin.
	DO_q_DrivetrainInverterTorqueless_DO AT %QX249.8: BOOL := FALSE;
	///Pin 1.32 - Digital input state for pin.
	DOS_q_DrivetrainInverterTorqueless_DO AT %IX770.12: BOOL := FALSE;
	///Pin 1.33 - Digital output status for output pin.
	DO_q_BatteryDischargePrecharge_DO AT %QX229.8: BOOL := FALSE;
	///Pin 1.33 - Digital input state for pin.
	DOS_q_BatteryDischargePrecharge_DO AT %IX770.10: BOOL := FALSE;
	///Pin 1.34 - Pulse ratio setting for PWFM channel [0..1000].
	PWFM_RATIO_u32_DynamoFrequency_PWFM AT %QB460: DWORD := 0;
	///Pin 1.34 - Frequency setting for PWFM channel [0..3000 Hz]
	PWFM_FREQ_u32_DynamoFrequency_PWFM AT %QB464: DWORD := 0;
	///Pin 1.35 - Digital output status for output pin.
	DO_q_Battery2ChargeMain_DO AT %QX219.8: BOOL := FALSE;
	///Pin 1.35 - Digital input state for pin.
	DOS_q_Battery2ChargeMain_DO AT %IX770.9: BOOL := FALSE;
	///Pin 2.6 - Filtered digital input status.
	DI_q_Battery1ChargeRq_DI: BOOL := FALSE;
	///Pin 2.7 - Filtered digital input status.
	DI_q_Battery1DiscahrgeRq_DI: BOOL := FALSE;
	///Pin 2.8 - Filtered digital input status.
	DI_q_Battery2ChargeRq_DI: BOOL := FALSE;
	///Pin 2.9 - Filtered digital input status.
	DI_q_Batter2DischargeRq_DI: BOOL := FALSE;
	///Pin 2.13 - Digital output status for output pin.
	DO_q_ChargePlugLockPulse_DO AT %QX119.8: BOOL := FALSE;
	///Pin 2.13 - Current feedback for output [0..2500 mA].
	PWFM_CM_q_ChargePlugLockPulse_DO AT %IB180: DWORD := 0;
	///Pin 2.13 - Digital input state for pin.
	DOS_q_ChargePlugLockPulse_DO AT %IX768.10: BOOL := FALSE;
	///Pin 2.13 - State of the overcurrent error.
	PWFM_OVERCURRENT_q_ChargePlugLockPulse_DO AT %IX94.12: BOOL := FALSE;
	///Pin 2.13 - State of the broken circuit error. Demands firmware version 1.2.X to work correctly. Not supported for step motor mode. For firmware versions for which brokent circuit is supported current limit can be set with function IO_PWFM_SET_BRK_DIAG_CURRENT.
	PWFM_OPENCIRCUIT_q_ChargePlugLockPulse_DO AT %IX94.14: BOOL := FALSE;
	///Pin 2.14 - Digital output status for output pin.
	DO_q_ChargePlugLockPosition_DO AT %QX109.8: BOOL := FALSE;
	///Pin 2.14 - Current feedback for output [0..2500 mA].
	PWFM_CM_q_ChargePlugLockPosition_DO AT %IB164: DWORD := 0;
	///Pin 2.14 - Digital input state for pin.
	DOS_q_ChargePlugLockPosition_DO AT %IX768.11: BOOL := FALSE;
	///Pin 2.14 - State of the overcurrent error.
	PWFM_OVERCURRENT_q_ChargePlugLockPosition_DO AT %IX86.12: BOOL := FALSE;
	///Pin 2.14 - State of the broken circuit error. Demands firmware version 1.2.X to work correctly. Not supported for step motor mode. For firmware versions for which brokent circuit is supported current limit can be set with function IO_PWFM_SET_BRK_DIAG_CURRENT.
	PWFM_OPENCIRCUIT_q_ChargePlugLockPosition_DO AT %IX86.14: BOOL := FALSE;
	///Pin 2.16 - Filtered digital input status.
	DI_q_ChargePlugLockStatus_DI: BOOL := FALSE;
	///Pin 2.23 - Filtered AI value
	AIPU_u16_HeaterDiagnose_AI: WORD := 0;
	///Pin 2.23 - Filtered AI value
	AI_u16_HeaterDiagnose_AI: WORD := 0;	
	///Pin 2.28 - Digital output status for output pin.
	DO_q_DrivetrainKL15D_DO AT %QX139.8: BOOL := FALSE;
	///Pin 2.28 - Current feedback for output [0..2500 mA].
	PWFM_CM_q_DrivetrainKL15D_DO AT %IB212: DWORD := 0;
	///Pin 2.28 - Digital input state for pin.
	DOS_q_DrivetrainKL15D_DO AT %IX768.12: BOOL := FALSE;
	///Pin 2.28 - State of the overcurrent error.
	PWFM_OVERCURRENT_q_DrivetrainKL15D_DO AT %IX110.12: BOOL := FALSE;
	///Pin 2.28 - State of the broken circuit error. Demands firmware version 1.2.X to work correctly. Not supported for step motor mode. For firmware versions for which brokent circuit is supported current limit can be set with function IO_PWFM_SET_BRK_DIAG_CURRENT.
	PWFM_OPENCIRCUIT_q_DrivetrainKL15D_DO AT %IX110.14: BOOL := FALSE;
	///Pin 2.29 - Digital output status for output pin.
	DO_q_DrivetrainKL15C_DO AT %QX129.8: BOOL := FALSE;
	///Pin 2.29 - Current feedback for output [0..2500 mA].
	PWFM_CM_q_DrivetrainKL15C_DO AT %IB196: DWORD := 0;
	///Pin 2.29 - Digital input state for pin.
	DOS_q_DrivetrainKL15C_DO AT %IX768.13: BOOL := FALSE;
	///Pin 2.29 - State of the overcurrent error.
	PWFM_OVERCURRENT_q_DrivetrainKL15C_DO AT %IX102.12: BOOL := FALSE;
	///Pin 2.29 - State of the broken circuit error. Demands firmware version 1.2.X to work correctly. Not supported for step motor mode. For firmware versions for which brokent circuit is supported current limit can be set with function IO_PWFM_SET_BRK_DIAG_CURRENT.
	PWFM_OPENCIRCUIT_q_DrivetrainKL15C_DO AT %IX102.14: BOOL := FALSE;
	///Pin 2.30 - Digital output status for output pin.
	DO_q_DrivetrainCoolingFan_DO AT %QX159.8: BOOL := FALSE;
	///Pin 2.30 - Current feedback for output [0..2500 mA].
	PWFM_CM_q_DrivetrainCoolingFan_DO AT %IB244: DWORD := 0;
	///Pin 2.30 - Digital input state for pin.
	DOS_q_DrivetrainCoolingFan_DO AT %IX768.14: BOOL := FALSE;
	///Pin 2.30 - State of the overcurrent error.
	PWFM_OVERCURRENT_q_DrivetrainCoolingFan_DO AT %IX126.12: BOOL := FALSE;
	///Pin 2.30 - State of the broken circuit error. Demands firmware version 1.2.X to work correctly. Not supported for step motor mode. For firmware versions for which brokent circuit is supported current limit can be set with function IO_PWFM_SET_BRK_DIAG_CURRENT.
	PWFM_OPENCIRCUIT_q_DrivetrainCoolingFan_DO AT %IX126.14: BOOL := FALSE;
	///Pin 2.31 - Digital output status for output pin.
	DO_q_DrievtrainPowerSteering_DO AT %QX149.8: BOOL := FALSE;
	///Pin 2.31 - Current feedback for output [0..2500 mA].
	PWFM_CM_q_DrievtrainPowerSteering_DO AT %IB228: DWORD := 0;
	///Pin 2.31 - Digital input state for pin.
	DOS_q_DrievtrainPowerSteering_DO AT %IX768.15: BOOL := FALSE;
	///Pin 2.31 - State of the overcurrent error.
	PWFM_OVERCURRENT_q_DrievtrainPowerSteering_DO AT %IX118.12: BOOL := FALSE;
	///Pin 2.31 - State of the broken circuit error. Demands firmware version 1.2.X to work correctly. Not supported for step motor mode. For firmware versions for which brokent circuit is supported current limit can be set with function IO_PWFM_SET_BRK_DIAG_CURRENT.
	PWFM_OPENCIRCUIT_q_DrievtrainPowerSteering_DO AT %IX118.14: BOOL := FALSE;
	///Pin 2.32 - Current feedback for output [0..2500 mA].
	PWFM_CM_u32_HeaterControl_PWFM AT %IB276: DWORD := 0;
	///Pin 2.32 - State of the overcurrent error.
	PWFM_OVERCURRENT_u32_HeaterControl_PWFM AT %IX142.12: BOOL := FALSE;
	///Pin 2.32 - State of the broken circuit error. Demands firmware version 1.2.X to work correctly. Not supported for step motor mode. For firmware versions for which brokent circuit is supported current limit can be set with function IO_PWFM_SET_BRK_DIAG_CURRENT.
	PWFM_OPENCIRCUIT_u32_HeaterControl_PWFM AT %IX142.14: BOOL := FALSE;
	///Pin 2.32 - Pulse ratio setting for PWFM channel [0..1000].
	PWFM_RATIO_u32_HeaterControl_PWFM AT %QB340: DWORD := 0;
	///Pin 2.32 - Frequency setting for PWFM channel [0..3000 Hz]
	PWFM_FREQ_u32_HeaterControl_PWFM AT %QB344: DWORD := 0;
	///Pin 2.33 - Digital output status for output pin.
	DO_q_DrievtrainAirCompressor_DO AT %QX169.8: BOOL := FALSE;
	///Pin 2.33 - Current feedback for output [0..2500 mA].
	PWFM_CM_q_DrievtrainAirCompressor_DO AT %IB260: DWORD := 0;
	///Pin 2.33 - Digital input state for pin.
	DOS_q_DrievtrainAirCompressor_DO AT %IX768.1: BOOL := FALSE;
	///Pin 2.33 - State of the overcurrent error.
	PWFM_OVERCURRENT_q_DrievtrainAirCompressor_DO AT %IX134.12: BOOL := FALSE;
	///Pin 2.33 - State of the broken circuit error. Demands firmware version 1.2.X to work correctly. Not supported for step motor mode. For firmware versions for which brokent circuit is supported current limit can be set with function IO_PWFM_SET_BRK_DIAG_CURRENT.
	PWFM_OPENCIRCUIT_q_DrievtrainAirCompressor_DO AT %IX134.14: BOOL := FALSE;
	///Pin 2.35 - Digital output state for sinking digital output.
	DO_q_DynamoD_DO AT %QX1408.11: BOOL := FALSE;
	///Pin 2.35 - Digital input state for pin.
	DOS_q_DynamoD_DO AT %IX770.6: BOOL := FALSE;
	///Pin 3.5 - Filtered digital input status.
	DI_q_DirectionSwitch_ReverseCrawl_DI: BOOL := FALSE;
	///Pin 3.6 - Filtered digital input status.
	DI_q_DirectionSwitch_Drive_DI: BOOL := FALSE;
	///Pin 3.7 - Filtered digital input status.
	DI_q_IlluminiationStatsus_DI: BOOL := FALSE;
	///Pin 3.8 - Filtered digital input status.
	DI_q_DirectionSwitch_Reverse_DI: BOOL := FALSE;
	///Pin 3.9 - Filtered digital input status.
	DI_q_DirectionSwitch_DriveCrawl_DI: BOOL := FALSE;
	///Pin 3.11 - Filtered digital input status.
	DI_q_DirectionSwitch_Neutral_DI: BOOL := FALSE;
	///Pin 3.12 - Filtered digital input status.
	DI_q_DoorOpen_DI: BOOL := FALSE;
	///Pin 3.14 - Filtered AI value
	AIPU_u16_HeaterDiagnose2_AI: WORD := 0;
	///Pin 3.14 - Filtered AI value
	AI_u16_HeaterDiagnose2_AI: WORD := 0;
	///Pin 3.15 - Filtered AI value
	AIPU_u16_VehicleThrottlePedal1_AI: WORD := 0;
	///Pin 3.15 - Filtered AI value
	AI_u16_VehicleThrottlePedal1_AI: WORD := 0;
	///Pin 3.16 - Filtered AI value for Pull-up measurement
	AIPU_u16_VehicleThrottlePedal2_AI: WORD := 0;
	///Pin 3.16 - Filtered AI value
	AI_u16_VehicleThrottlePedal2_AI: WORD := 0;
	///Pin 3.22 - Filtered digital input status.
	DI_q_VehicleKL15_DI: BOOL := FALSE;
	///Pin 3.23 - Filtered digital input status.
	DI_q_VehicleKL51_DI: BOOL := FALSE;
	///Pin 3.26 - Digital output status for output pin.
	DO_q_ChargersWakeup_DO AT %QX199.8: BOOL := FALSE;
	///Pin 3.26 - Current feedback for output [0..2500 mA].
	PWFM_CM_q_ChargersWakeup_DO AT %IB308: DWORD := 0;
	///Pin 3.26 - Digital input state for pin.
	DOS_q_ChargersWakeup_DO AT %IX768.2: BOOL := FALSE;
	///Pin 3.26 - State of the overcurrent error.
	PWFM_OVERCURRENT_q_ChargersWakeup_DO AT %IX158.12: BOOL := FALSE;
	///Pin 3.26 - State of the broken circuit error. Demands firmware version 1.2.X to work correctly. Not supported for step motor mode. For firmware versions for which brokent circuit is supported current limit can be set with function IO_PWFM_SET_BRK_DIAG_CURRENT.
	PWFM_OPENCIRCUIT_q_ChargersWakeup_DO AT %IX158.14: BOOL := FALSE;
	///Pin 3.27 - Digital output status for output pin.
	DO_q_DashboardDCDCStatus_DO AT %QX189.8: BOOL := FALSE;
	///Pin 3.27 - Current feedback for output [0..2500 mA].
	PWFM_CM_q_DashboardDCDCStatus_DO AT %IB292: DWORD := 0;
	///Pin 3.27 - Digital input state for pin.
	DOS_q_DashboardDCDCStatus_DO AT %IX768.3: BOOL := FALSE;
	///Pin 3.27 - State of the overcurrent error.
	PWFM_OVERCURRENT_q_DashboardDCDCStatus_DO AT %IX150.12: BOOL := FALSE;
	///Pin 3.27 - State of the broken circuit error. Demands firmware version 1.2.X to work correctly. Not supported for step motor mode. For firmware versions for which brokent circuit is supported current limit can be set with function IO_PWFM_SET_BRK_DIAG_CURRENT.
	PWFM_OPENCIRCUIT_q_DashboardDCDCStatus_DO AT %IX150.14: BOOL := FALSE;
	///Pin 3.28 - Filtered digital input status.
	DI_q_HeaterIn_DI: BOOL := FALSE;
	///Pin 3.29 - Digital output status for output pin.
	DO_q_HeaterOut_DI AT %QX9.8: BOOL := FALSE;
	///Pin 3.29 - Current feedback for output [0..2500 mA].
	PWFM_CM_q_HeaterOut_DI AT %IB4: DWORD := 0;
	///Pin 3.29 - Digital input state for pin.
	DOS_q_HeaterOut_DI AT %IX768.5: BOOL := FALSE;
	///Pin 3.29 - State of the overcurrent error.
	PWFM_OVERCURRENT_q_HeaterOut_DI AT %IX6.12: BOOL := FALSE;
	///Pin 3.29 - State of the broken circuit error. Demands firmware version 1.2.X to work correctly. Not supported for step motor mode. For firmware versions for which brokent circuit is supported current limit can be set with function IO_PWFM_SET_BRK_DIAG_CURRENT.
	PWFM_OPENCIRCUIT_q_HeaterOut_DI AT %IX6.14: BOOL := FALSE;
	///Pin 3.29 - Filtered Voltage measurement value for output pin  [10 mV].
	AI_q_HeaterOut_DI_Ai: WORD := 0;
	///Pin 3.30 - Digital output status for output pin.
	DO_q_DrivetrainInverterRf1_DO AT %QX39.8: BOOL := FALSE;
	///Pin 3.30 - Current feedback for output [0..2500 mA].
	PWFM_CM_q_DrivetrainInverterRf1_DO AT %IB52: DWORD := 0;
	///Pin 3.30 - Digital input state for pin.
	DOS_q_DrivetrainInverterRf1_DO AT %IX768.6: BOOL := FALSE;
	///Pin 3.30 - State of the overcurrent error.
	PWFM_OVERCURRENT_q_DrivetrainInverterRf1_DO AT %IX30.12: BOOL := FALSE;
	///Pin 3.30 - State of the broken circuit error. Demands firmware version 1.2.X to work correctly. Not supported for step motor mode. For firmware versions for which brokent circuit is supported current limit can be set with function IO_PWFM_SET_BRK_DIAG_CURRENT.
	PWFM_OPENCIRCUIT_q_DrivetrainInverterRf1_DO AT %IX30.14: BOOL := FALSE;
	///Pin 3.30 - Filtered Voltage measurement value for output pin  [10 mV].
	AI_q_DrivetrainInverterRf1_DO_Ai: WORD := 0;
	///Pin 3.31 - Digital output status for output pin.
	DO_q_DrivetrainInverterRf2_DO AT %QX29.8: BOOL := FALSE;
	///Pin 3.31 - Current feedback for output [0..2500 mA].
	PWFM_CM_q_DrivetrainInverterRf2_DO AT %IB36: DWORD := 0;
	///Pin 3.31 - Digital input state for pin.
	DOS_q_DrivetrainInverterRf2_DO AT %IX768.7: BOOL := FALSE;
	///Pin 3.31 - State of the overcurrent error.
	PWFM_OVERCURRENT_q_DrivetrainInverterRf2_DO AT %IX22.12: BOOL := FALSE;
	///Pin 3.31 - State of the broken circuit error. Demands firmware version 1.2.X to work correctly. Not supported for step motor mode. For firmware versions for which brokent circuit is supported current limit can be set with function IO_PWFM_SET_BRK_DIAG_CURRENT.
	PWFM_OPENCIRCUIT_q_DrivetrainInverterRf2_DO AT %IX22.14: BOOL := FALSE;
	///Pin 3.31 - Filtered Voltage measurement value for output pin  [10 mV].
	AI_q_DrivetrainInverterRf2_DO_Ai: WORD := 0;
	///Pin 3.32 - Digital output status for output pin.
	DO_q_DrivetrainDCDCInhibit_DO AT %QX59.8: BOOL := FALSE;
	///Pin 3.32 - Current feedback for output [0..2500 mA].
	PWFM_CM_q_DrivetrainDCDCInhibit_DO AT %IB84: DWORD := 0;
	///Pin 3.32 - Digital input state for pin.
	DOS_q_DrivetrainDCDCInhibit_DO AT %IX770.1: BOOL := FALSE;
	///Pin 3.32 - State of the overcurrent error.
	PWFM_OVERCURRENT_q_DrivetrainDCDCInhibit_DO AT %IX46.12: BOOL := FALSE;
	///Pin 3.32 - State of the broken circuit error. Demands firmware version 1.2.X to work correctly. Not supported for step motor mode. For firmware versions for which brokent circuit is supported current limit can be set with function IO_PWFM_SET_BRK_DIAG_CURRENT.
	PWFM_OPENCIRCUIT_q_DrivetrainDCDCInhibit_DO AT %IX46.14: BOOL := FALSE;
	///Pin 3.32 - Filtered Voltage measurement value for output pin  [10 mV].
	AI_q_DrivetrainDCDCInhibit_DO_Ai: WORD := 0;
	///Pin 3.33 - Digital output status for output pin.
	DO_q_ChargePlugLED_Green_DO AT %QX49.8: BOOL := FALSE;
	///Pin 3.33 - Current feedback for output [0..2500 mA].
	PWFM_CM_q_ChargePlugLED_Green_DO AT %IB68: DWORD := 0;
	///Pin 3.33 - Digital input state for pin.
	DOS_q_ChargePlugLED_Green_DO AT %IX770.0: BOOL := FALSE;
	///Pin 3.33 - State of the overcurrent error.
	PWFM_OVERCURRENT_q_ChargePlugLED_Green_DO AT %IX38.12: BOOL := FALSE;
	///Pin 3.33 - State of the broken circuit error. Demands firmware version 1.2.X to work correctly. Not supported for step motor mode. For firmware versions for which brokent circuit is supported current limit can be set with function IO_PWFM_SET_BRK_DIAG_CURRENT.
	PWFM_OPENCIRCUIT_q_ChargePlugLED_Green_DO AT %IX38.14: BOOL := FALSE;
	///Pin 3.33 - Filtered Voltage measurement value for output pin  [10 mV].
	AI_q_ChargePlugLED_Green_DO_Ai: WORD := 0;
	///Pin 3.34 - Digital output status for output pin.
	DO_q_ChargePlugLED_Blue_DO AT %QX79.8: BOOL := FALSE;
	///Pin 3.34 - Current feedback for output [0..2500 mA].
	PWFM_CM_q_ChargePlugLED_Blue_DO AT %IB116: DWORD := 0;
	///Pin 3.34 - Digital input state for pin.
	DOS_q_ChargePlugLED_Blue_DO AT %IX770.3: BOOL := FALSE;
	///Pin 3.34 - State of the overcurrent error.
	PWFM_OVERCURRENT_q_ChargePlugLED_Blue_DO AT %IX62.12: BOOL := FALSE;
	///Pin 3.34 - State of the broken circuit error. Demands firmware version 1.2.X to work correctly. Not supported for step motor mode. For firmware versions for which brokent circuit is supported current limit can be set with function IO_PWFM_SET_BRK_DIAG_CURRENT.
	PWFM_OPENCIRCUIT_q_ChargePlugLED_Blue_DO AT %IX62.14: BOOL := FALSE;
	///Pin 3.34 - Filtered Voltage measurement value for output pin  [10 mV].
	AI_q_ChargePlugLED_Blue_DO_Ai: WORD := 0;
	///Pin 3.35 - Digital output status for output pin.
	DO_q_ChargePlugLED_Red_DO AT %QX69.8: BOOL := FALSE;
	///Pin 3.35 - Current feedback for output [0..2500 mA].
	PWFM_CM_q_ChargePlugLED_Red_DO AT %IB100: DWORD := 0;
	///Pin 3.35 - Digital input state for pin.
	DOS_q_ChargePlugLED_Red_DO AT %IX770.2: BOOL := FALSE;
	///Pin 3.35 - State of the overcurrent error.
	PWFM_OVERCURRENT_q_ChargePlugLED_Red_DO AT %IX54.12: BOOL := FALSE;
	///Pin 3.35 - State of the broken circuit error. Demands firmware version 1.2.X to work correctly. Not supported for step motor mode. For firmware versions for which brokent circuit is supported current limit can be set with function IO_PWFM_SET_BRK_DIAG_CURRENT.
	PWFM_OPENCIRCUIT_q_ChargePlugLED_Red_DO AT %IX54.14: BOOL := FALSE;
	///Pin 3.35 - Filtered Voltage measurement value for output pin  [10 mV].
	AI_q_ChargePlugLED_Red_DO_Ai: WORD := 0;
END_VAR

// Application/CodeTemplate/Globals/IO_CONFIG
VAR_GLOBAL
	///Pin 1.9 - Enables 10 V pull-up for pin.
	AI_SET_PU_u16_DrivetrainTemp_AI AT %QX1411.12: BOOL := FALSE;
	///Pin 1.9 - Signal area selection mA/V.
	AI_SET_mA_u16_DrivetrainTemp_AI AT %QX1411.13: BOOL := FALSE;
	///Pin 1.10 - Enables 10 V pull-up for pin.
	AI_SET_PU_u16_ChargePlugPresent_AI AT %QX1411.14: BOOL := FALSE;
	///Pin 1.10 - Signal area selection mA/V.
	AI_SET_mA_u16_ChargePlugPresent_AI AT %QX1411.15: BOOL := FALSE;
	///Pin 1.11 - Variable notifies possible configuration error code.
	PI_INIT_ERROR_q_BatteryInterlockIn_DI: DINT := 0;
	///Pin 1.12 - Possible init error for PWFM channel init (0 = Success).
	PWFM_ERROR_INIT_q_BackupPump_DO: DINT := 0;
	///Pin 1.12 - Used mode for PWFM channel.
	PWFM_MODE_q_BackupPump_DO AT %IB128: DWORD := 0;
	///Pin 1.20 - Pull-up enable selection for pin.
	AI_SET_PU_u16_Heater1Temperature_AI AT %QX1411.0: BOOL := FALSE;
	///Pin 1.20 - Signal area selection mA/V.
	AI_SET_mA_u16_Heater1Temperature_AI AT %QX1411.1: BOOL := FALSE;
	///Pin 1.21 - Pull-up enable selection for pin.
	AI_SET_PU_u16_Heater2Temperature_AI AT %QX1411.2: BOOL := FALSE;
	///Pin 1.21 - Signal area selection mA/V.
	AI_SET_mA_u16_Heater2Temperature_AI AT %QX1411.3: BOOL := FALSE;
	///Pin 1.22 - Possible init error for PWFM channel init (0 = Success).
	PWFM_ERROR_INIT_q_BatteryDischargeMain_DO: DINT := 0;
	///Pin 1.22 - Used mode for PWFM channel.
	PWFM_MODE_q_BatteryDischargeMain_DO AT %IB320: DWORD := 0;
	///Pin 1.23 - Possible init error for PWFM channel init (0 = Success).
	PWFM_ERROR_INIT_q_AirPressureReliefValve_DO: DINT := 0;
	///Pin 1.23 - Used mode for PWFM channel.
	PWFM_MODE_q_AirPressureReliefValve_DO AT %IB144: DWORD := 0;
	///Pin 1.29 - Possible init error for PWFM channel init (0 = Success).
	PWFM_ERROR_INIT_q_Battery1ChargePrecharge_DO: DINT := 0;
	///Pin 1.29 - Used mode for PWFM channel.
	PWFM_MODE_q_Battery1ChargePrecharge_DO AT %IB432: DWORD := 0;
	///Pin 1.30 - Possible init error for PWFM channel init (0 = Success).
	PWFM_ERROR_INIT_q_Battery1ChargeMain_DO: DINT := 0;
	///Pin 1.30 - Used mode for PWFM channel.
	PWFM_MODE_q_Battery1ChargeMain_DO AT %IB416: DWORD := 0;
	///Pin 1.31 - Possible init error for PWFM channel init (0 = Success).
	PWFM_ERROR_INIT_q_Battery2ChargePrecharge_DO: DINT := 0;
	///Pin 1.31 - Used mode for PWFM channel.
	PWFM_MODE_q_Battery2ChargePrecharge_DO AT %IB400: DWORD := 0;
	///Pin 1.32 - Possible init error for PWFM channel init (0 = Success).
	PWFM_ERROR_INIT_q_DrivetrainInverterTorqueless_DO: DINT := 0;
	///Pin 1.32 - Used mode for PWFM channel.
	PWFM_MODE_q_DrivetrainInverterTorqueless_DO AT %IB384: DWORD := 0;
	///Pin 1.33 - Possible init error for PWFM channel init (0 = Success).
	PWFM_ERROR_INIT_q_BatteryDischargePrecharge_DO: DINT := 0;
	///Pin 1.33 - Used mode for PWFM channel.
	PWFM_MODE_q_BatteryDischargePrecharge_DO AT %IB352: DWORD := 0;
	///Pin 1.34 - Possible init error for PWFM channel init (0 = Success).
	PWFM_ERROR_INIT_u32_DynamoFrequency_PWFM: DINT := 0;
	///Pin 1.34 - Used mode for PWFM channel.
	PWFM_MODE_u32_DynamoFrequency_PWFM AT %IB368: DWORD := 0;
	///Pin 1.35 - Possible init error for PWFM channel init (0 = Success).
	PWFM_ERROR_INIT_q_Battery2ChargeMain_DO: DINT := 0;
	///Pin 1.35 - Used mode for PWFM channel.
	PWFM_MODE_q_Battery2ChargeMain_DO AT %IB336: DWORD := 0;
	///Pin 2.6 - Variable notifies possible configuration error code.
	PI_INIT_ERROR_q_Battery1ChargeRq_DI: DINT := 0;
	///Pin 2.7 - Variable notifies possible configuration error code.
	PI_INIT_ERROR_q_Battery1DiscahrgeRq_DI: DINT := 0;
	///Pin 2.8 - Variable notifies possible configuration error code.
	PI_INIT_ERROR_q_Battery2ChargeRq_DI: DINT := 0;
	///Pin 2.9 - Variable notifies possible configuration error code.
	PI_INIT_ERROR_q_Batter2DischargeRq_DI: DINT := 0;
	///Pin 2.13 - Possible init error for PWFM channel init (0 = Success).
	PWFM_ERROR_INIT_q_ChargePlugLockPulse_DO: DINT := 0;
	///Pin 2.13 - Used mode for PWFM channel.
	PWFM_MODE_q_ChargePlugLockPulse_DO AT %IB176: DWORD := 0;
	///Pin 2.14 - Possible init error for PWFM channel init (0 = Success).
	PWFM_ERROR_INIT_q_ChargePlugLockPosition_DO: DINT := 0;
	///Pin 2.14 - Used mode for PWFM channel.
	PWFM_MODE_q_ChargePlugLockPosition_DO AT %IB160: DWORD := 0;
	///Pin 2.23 - Pull-up enable selection for pin.
	AI_SET_PU_u16_HeaterDiagnose_AI AT %QX1411.4: BOOL := FALSE;
	///Pin 2.23 - Signal area selection mA/V.
	AI_SET_mA_u16_HeaterDiagnose_AI AT %QX1411.5: BOOL := FALSE;
	///Pin 2.28 - Possible init error for PWFM channel init (0 = Success).
	PWFM_ERROR_INIT_q_DrivetrainKL15D_DO: DINT := 0;
	///Pin 2.28 - Used mode for PWFM channel.
	PWFM_MODE_q_DrivetrainKL15D_DO AT %IB208: DWORD := 0;
	///Pin 2.29 - Possible init error for PWFM channel init (0 = Success).
	PWFM_ERROR_INIT_q_DrivetrainKL15C_DO: DINT := 0;
	///Pin 2.29 - Used mode for PWFM channel.
	PWFM_MODE_q_DrivetrainKL15C_DO AT %IB192: DWORD := 0;
	///Pin 2.30 - Possible init error for PWFM channel init (0 = Success).
	PWFM_ERROR_INIT_q_DrivetrainCoolingFan_DO: DINT := 0;
	///Pin 2.30 - Used mode for PWFM channel.
	PWFM_MODE_q_DrivetrainCoolingFan_DO AT %IB240: DWORD := 0;
	///Pin 2.31 - Possible init error for PWFM channel init (0 = Success).
	PWFM_ERROR_INIT_q_DrievtrainPowerSteering_DO: DINT := 0;
	///Pin 2.31 - Used mode for PWFM channel.
	PWFM_MODE_q_DrievtrainPowerSteering_DO AT %IB224: DWORD := 0;
	///Pin 2.32 - Possible init error for PWFM channel init (0 = Success).
	PWFM_ERROR_INIT_u32_HeaterControl_PWFM: DINT := 0;
	///Pin 2.32 - Used mode for PWFM channel.
	PWFM_MODE_u32_HeaterControl_PWFM AT %IB272: DWORD := 0;
	///Pin 2.33 - Possible init error for PWFM channel init (0 = Success).
	PWFM_ERROR_INIT_q_DrievtrainAirCompressor_DO: DINT := 0;
	///Pin 2.33 - Used mode for PWFM channel.
	PWFM_MODE_q_DrievtrainAirCompressor_DO AT %IB256: DWORD := 0;
	///Pin 3.5 - Variable notifies possible configuration error code.
	PI_INIT_ERROR_q_DirectionSwitch_ReverseCrawl_DI: DINT := 0;
	///Pin 3.6 - Variable notifies possible configuration error code.
	PI_INIT_ERROR_q_DirectionSwitch_Drive_DI: DINT := 0;
	///Pin 3.8 - Variable notifies possible configuration error code.
	PI_INIT_ERROR_q_DirectionSwitch_Reverse_DI: DINT := 0;
	///Pin 3.9 - Variable notifies possible configuration error code.
	PI_INIT_ERROR_q_DirectionSwitch_DriveCrawl_DI: DINT := 0;
	///Pin 3.11 - Variable notifies possible configuration error code.
	PI_INIT_ERROR_q_DirectionSwitch_Neutral_DI: DINT := 0;
	///Pin 3.12 - Variable notifies possible configuration error code.
	PI_INIT_ERROR_q_DoorOpen_DI: DINT := 0;
	///Pin 3.14 - Pull-up enable selection for pin.
	AI_SET_PU_u16_HeaterDiagnose2_AI AT %QX1410.0: BOOL := FALSE;
	///Pin 3.14 - Signal area selection mA/V.
	AI_SET_mA_u16_HeaterDiagnose2_AI AT %QX1410.1: BOOL := FALSE;
	///Pin 3.15 - Pull-up enable selection for pin.
	AI_SET_PU_u16_VehicleThrottlePedal1_AI AT %QX1410.2: BOOL := FALSE;
	///Pin 3.15 - Signal area selection mA/V.
	AI_SET_mA_u16_VehicleThrottlePedal1_AI AT %QX1410.3: BOOL := FALSE;
	///Pin 3.16 - Pull-up enable selection for pin.
	AI_SET_PU_u16_VehicleThrottlePedal2_AI AT %QX1410.4: BOOL := FALSE;
	///Pin 3.16 - Signal area selection mA/V.
	AI_SET_mA_u16_VehicleThrottlePedal2_AI AT %QX1410.5: BOOL := FALSE;
	///Pin 3.22 - Variable notifies possible configuration error code.
	PI_INIT_ERROR_q_VehicleKL15_DI: DINT := 0;
	///Pin 3.23 - Variable notifies possible configuration error code.
	PI_INIT_ERROR_q_VehicleKL51_DI: DINT := 0;
	///Pin 3.26 - Possible init error for PWFM channel init (0 = Success).
	PWFM_ERROR_INIT_q_ChargersWakeup_DO: DINT := 0;
	///Pin 3.26 - Used mode for PWFM channel.
	PWFM_MODE_q_ChargersWakeup_DO AT %IB304: DWORD := 0;
	///Pin 3.27 - Possible init error for PWFM channel init (0 = Success).
	PWFM_ERROR_INIT_q_DashboardDCDCStatus_DO: DINT := 0;
	///Pin 3.27 - Used mode for PWFM channel.
	PWFM_MODE_q_DashboardDCDCStatus_DO AT %IB288: DWORD := 0;
	///Pin 3.28 - Possible init error for PWFM channel init (0 = Success).
	PWFM_ERROR_INIT_q_HeaterIn_DI: DINT := 0;
	///Pin 3.29 - Possible init error for PWFM channel init (0 = Success).
	PWFM_ERROR_INIT_q_HeaterOut_DI: DINT := 0;
	///Pin 3.29 - Used mode for PWFM channel.
	PWFM_MODE_q_HeaterOut_DI AT %IB0: DWORD := 0;
	///Pin 3.30 - Possible init error for PWFM channel init (0 = Success).
	PWFM_ERROR_INIT_q_DrivetrainInverterRf1_DO: DINT := 0;
	///Pin 3.30 - Used mode for PWFM channel.
	PWFM_MODE_q_DrivetrainInverterRf1_DO AT %IB48: DWORD := 0;
	///Pin 3.31 - Possible init error for PWFM channel init (0 = Success).
	PWFM_ERROR_INIT_q_DrivetrainInverterRf2_DO: DINT := 0;
	///Pin 3.31 - Used mode for PWFM channel.
	PWFM_MODE_q_DrivetrainInverterRf2_DO AT %IB32: DWORD := 0;
	///Pin 3.32 - Possible init error for PWFM channel init (0 = Success).
	PWFM_ERROR_INIT_q_DrivetrainDCDCInhibit_DO: DINT := 0;
	///Pin 3.32 - Used mode for PWFM channel.
	PWFM_MODE_q_DrivetrainDCDCInhibit_DO AT %IB80: DWORD := 0;
	///Pin 3.33 - Possible init error for PWFM channel init (0 = Success).
	PWFM_ERROR_INIT_q_ChargePlugLED_Green_DO: DINT := 0;
	///Pin 3.33 - Used mode for PWFM channel.
	PWFM_MODE_q_ChargePlugLED_Green_DO AT %IB64: DWORD := 0;
	///Pin 3.34 - Possible init error for PWFM channel init (0 = Success).
	PWFM_ERROR_INIT_q_ChargePlugLED_Blue_DO: DINT := 0;
	///Pin 3.34 - Used mode for PWFM channel.
	PWFM_MODE_q_ChargePlugLED_Blue_DO AT %IB112: DWORD := 0;
	///Pin 3.35 - Possible init error for PWFM channel init (0 = Success).
	PWFM_ERROR_INIT_q_ChargePlugLED_Red_DO: DINT := 0;
	///Pin 3.35 - Used mode for PWFM channel.
	PWFM_MODE_q_ChargePlugLED_Red_DO AT %IB96: DWORD := 0;
	///Pin 1000.100 - Pull-up configuration for pins 1.22 and 1.35
	PWFM_SET_PU_1_22_and_1_35 AT %QX1410.12: BOOL := FALSE;
	///Pin 1000.100 - Pull-up configuration for pins 1.33 and 1.34
	PWFM_SET_PU_1_33_and_1_34 AT %QX1410.13: BOOL := FALSE;
	///Pin 1000.100 - Pull-up configuration for pins 1.31 and 1.32
	PWFM_SET_PU_1_31_and_1_32 AT %QX1410.14: BOOL := FALSE;
	///Pin 1000.100 - Pull-up configuration for pins 1.29 and 1.30
	PWFM_SET_PU_1_29_and_1_30 AT %QX1410.15: BOOL := FALSE;
	///Pin 1000.100 - Pull-up configuration for pins 2.6 and 2.7
	PI_SET_PU_2_06_and_2_07 AT %QX1410.8: BOOL := FALSE;
	///Pin 1000.100 - Pull-up configuration for pins 2.8 and 2.9.
	PI_SET_PU_2_08_and_2_09 AT %QX1410.10: BOOL := FALSE;
	///Pin 1000.100 - Pull-up configuration for pins 3.5 and 3.6.
	PI_SET_PU_3_05_and_3_06 AT %QX1412.10: BOOL := FALSE;
	///Pin 1000.100 - Pull-up configuration for pins 3.8 and 3.9
	PI_SET_PU_3_08_and_3_09 AT %QX1412.8: BOOL := FALSE;
	///Pin 1000.100 - Pull-up configuration for pins 3.11 and 3.12
	PI_SET_PU_3_11_and_3_12 AT %QX1412.9: BOOL := FALSE;
	///Pin 1000.100 - Pull-up configuration for pins 3.21 and 3.22
	PI_SET_PU_3_21_and_3_22 AT %QX1412.11: BOOL := FALSE;
	///Pin 1000.100 - Pull-up configuration for pins 1.11 and 3.23
	PI_SET_PU_1_11_and_3_23 AT %QX1412.12: BOOL := FALSE;
	///Pin 1000.100 - Pull-up configuration for pins 2.16 and 2.17
	PI_SET_PU_2_16_and_2_17 AT %QX1411.6: BOOL := FALSE;
	///Pin 1000.100 - Pull-up configuration for pins 2.19 and 2.20
	PI_SET_PU_2_19_and_2_20 AT %QX1411.7: BOOL := FALSE;
	///Pin 1000.101 - Used voltage range. Range configuration for pins 2.6 and 2.7
	PI_SET_RANGE_2_06_and_2_07 AT %QX1410.9: BOOL := FALSE;
	///Pin 1000.101 - Used voltage range. Range configuration for pins 2.8 and 2.9.
	PI_SET_RANGE_2_08_and_2_09 AT %QX1410.11: BOOL := FALSE;
	///Pin 1000.102 - System supply voltage level [24 V]
	G_SupplyVoltageLevel: WORD := 24;
END_VAR

// Application/CodeTemplate/Globals/IO_INTERNAL
VAR_GLOBAL
	///Filtered supply logic raw value (10 sample mean).
	AI_SupplyLogic: WORD := 0;
	///Logic voltage [10 mV].
	SUPPLY_Logic: WORD := 0;
	///Disable/Enable power switch 1.
	POWER_1_Enable: BOOL := FALSE;
	///Filtered Power switch 1 voltage raw value (10 sample mean).
	AI_SupplyPower1: WORD := 0;
	///Power switch 1 voltage [10 mV].
	SUPPLY_Power1: WORD := 0;
	///Disable/Enable power switch 2.
	POWER_2_Enable: BOOL := FALSE;
	///Filtered Power switch 2 voltage raw value (10 sample mean).
	AI_SupplyPower2: WORD := 0;
	///Power switch 2 voltage [10 mV].
	SUPPLY_Power2: WORD := 0;
	///Enable for 5 V reference.
	REF_OUT_5V_Enable AT %QX1412.14: BOOL := FALSE;
	///Filtered Ref 5 V voltage raw value (10 sample mean).
	AI_Ref5V: WORD := 0;
	///Scaled Ref 5 V voltage  [10 mV].
	REF_5V: WORD := 0;
	///Enable for 10 V reference.
	REF_OUT_10V_Enable AT %QX1412.13: BOOL := FALSE;
	///Filtered Ref 10 V voltage raw value (10 sample mean).
	AI_Ref10V: WORD := 0;
	///Scaled Ref 10 V voltage [10 mV].
	REF_10V: WORD := 0;
	///Filtered 10 V Pull-ups voltage raw value (10 sample mean).
	AI_10VPullUpSupply: WORD := 0;
	///Scaled 10 V Pull-ups voltage [10 mV].
	REF_10VPullUpSupply: WORD := 0;
	///Filtered ADC reference. raw value (10 sample mean).
	AI_InternADCReference: WORD := 0;
	///ADC reference voltage [10 mV].
	REF_InternADC: WORD := 0;
	///Filtered PCB temperature raw value (10 sample mean).
	AI_PCBTemperature: WORD := 0;
	///PCB temperature [0.1 C].
	TEMP_PCB: INT := 0;
	///Filtered core temperature raw value (10 sample mean).
	AI_CoreTemperature: WORD := 0;
	///Core temperature [0.1 C].
	TEMP_CoreTemperature: INT := 0;
	///Filtered pin 2.24 / 2.25 input voltage value.
	AI_Power1Pin: WORD := 0;
	///Scaled pin 2.24 / 2.25 input voltage value [0.01 V]
	SUPPLY_Power1Pin: WORD := 0;
	///Filtered pin 3.24 / 3.25 input voltage value.
	AI_Power2Pin: WORD := 0;
	///Scaled pin 3.24 / 3.25 input voltage value [0.01 V]
	SUPPLY_Power2Pin: WORD := 0;
	///Pin 2.16 - Variable notifies possible configuration error code.
	PI_ERROR_q_ChargePlugLockStatus_DI: DINT := 0;
	///Pin 3.7 - Variable notifies possible configuration error code.
	PI_ERROR_q_IlluminiationStatsus_DI: DINT := 0;
END_VAR

// Application/CodeTemplate/Globals/IO_RAW
VAR_GLOBAL
	///Error field for AI Errors.
	AI_ERRORS AT %IW2048: WORD := 0;
	///General time stamp array for ADC conversions.
	AI_ARR_TS AT %IW2226: ARRAY [1..50] OF WORD;
	///Index for place in latest conversion in conversion arrays.
	AI_ARR_INDEX AT %IB4099: BYTE := 0;
	///Latest measured raw value for logic supply.
	AI_RAW_SupplyLogic AT %IW2093: WORD := 0;
	///Array of  measured raw values for logic supply.
	AI_ARR_SupplyLogic AT %IW4026: ARRAY [1..50] OF WORD;
	///Latest measured raw value for Power supply 1.
	AI_RAW_SupplyPower1 AT %IW2095: WORD := 0;
	///Array of  measured raw values for power switch 1.
	AI_ARR_SupplyPower1 AT %IW4126: ARRAY [1..50] OF WORD;
	///Latest measured raw value for Power supply 2.
	AI_RAW_SupplyPower2 AT %IW2064: WORD := 0;
	///Array of  measured raw values for power switch 2.
	AI_ARR_SupplyPower2 AT %IW2576: ARRAY [1..50] OF WORD;
	///Latest measured raw value for Ref 5 V voltage.
	AI_RAW_Ref5V AT %IW2070: WORD := 0;
	///Array of  measured raw values for Ref 5 V voltage.
	AI_ARR_Ref5V AT %IW2876: ARRAY [1..50] OF WORD;
	///Latest measured raw value for Ref 10 V voltage.
	AI_RAW_Ref10V AT %IW2072: WORD := 0;
	///Array of  measured raw values for Ref 10 V voltage.
	AI_ARR_Ref10V AT %IW2976: ARRAY [1..50] OF WORD;
	///Latest measured raw value for 10 V Pull-ups voltage.
	AI_RAW_10VPullUpSupply AT %IW2074: WORD := 0;
	///Array of  measured raw values for 10 V Pull-ups voltage.
	AI_ARR_10VPullUpSupply AT %IW3076: ARRAY [1..50] OF WORD;
	///Latest measured raw value for ADC reference.
	AI_RAW_InternADCReference AT %IW2068: WORD := 0;
	///Array of  measured raw values for ADC reference.
	AI_ARR_InternADCReference AT %IW2776: ARRAY [1..50] OF WORD;
	///Latest measured raw value for PCB temperature.
	AI_RAW_PCBTemperature AT %IW2066: WORD := 0;
	///Array of  measured raw values for PCB temperture.
	AI_ARR_PCBTemperature AT %IW2676: ARRAY [1..50] OF WORD;
	///Latest measured raw value for PCB temperature.
	AI_RAW_CoreTemperature AT %IW2076: WORD := 0;
	///Array of measured raw values for PCB temperture.
	AI_ARR_CoreTemperature AT %IW3176: ARRAY [1..50] OF WORD;
	///Latest measured value for voltage in pin 2.24 / 2.25.
	AI_RAW_Power1Pin AT %IW2096: WORD := 0;
	///Array of  measured raw values for voltage in  pin 2.24 / 2.25.
	AI_ARR_Power1Pin  AT %IW4176: ARRAY [1..50] OF WORD;
	///Latest measured value for voltage in pin 3.24 / 3.25.
	AI_RAW_Power2Pin AT %IW2097: WORD := 0;
	///Array of  measured raw values for voltage in  pin 3.24 / 3.25.
	AI_ARR_Power2Pin  AT %IW4226: ARRAY [1..50] OF WORD;
	///Pin 1.9 - Latest measurement value for pin's input signal.
	AI_RAW_u16_DrivetrainTemp_AI AT %IW2056: WORD := 0;
	///Pin 1.9 - Array of 50 latest conversion values for pin's input signal.
	AI_ARR_u16_DrivetrainTemp_AI AT %IW2176: ARRAY [1..50] OF WORD;
	///Pin 1.9 - Latest measurement value for pin's pull-up voltage.
	AIPU_RAW_u16_DrivetrainTemp_AI AT %IW2065: WORD := 0;
	///Pin 1.9 - Array of 50 latest conversion values for pin's pull-up voltage.
	AIPU_ARR_u16_DrivetrainTemp_AI AT %IW2626: ARRAY [1..50] OF WORD;
	///Pin 1.10 - Latest measurement value for pin's input signal.
	AI_RAW_u16_ChargePlugPresent_AI AT %IW2077: WORD := 0;
	///Pin 1.10 - Array of 50 latest conversion values for pin's input signal.
	AI_ARR_u16_ChargePlugPresent_AI AT %IW3226: ARRAY [1..50] OF WORD;
	///Pin 1.10 - Latest measurement value for pin's pull-up voltage.
	AIPU_RAW_u16_ChargePlugPresent_AI AT %IW2067: WORD := 0;
	///Pin 1.10 - Array of 50 latest conversion values for pin's pull-up voltage.
	AIPU_ARR_u16_ChargePlugPresent_AI AT %IW2726: ARRAY [1..50] OF WORD;
	///Pin 1.11 - Unfiltered digital input status.
	DI_RAW_q_BatteryInterlockIn_DI AT %IX1030.8: BOOL := FALSE;
	///Pin 1.20 - Latest measurement value for pin's input signal.
	AI_RAW_u16_Heater1Temperature_AI AT %IW2058: WORD := 0;
	///Pin 1.20 - Array of 50 latest conversion values for pin's input signal.
	AI_ARR_u16_Heater1Temperature_AI AT %IW2276: ARRAY [1..50] OF WORD;
	///Pin 1.20 - Latest measurement value for pin's pull-up voltage.
	AIPU_RAW_u16_Heater1Temperature_AI AT %IW2069: WORD := 0;
	///Pin 1.20 - Array of 50 latest conversion values for pin's pull-up voltage.
	AIPU_ARR_u16_Heater1Temperature_AI AT %IW2826: ARRAY [1..50] OF WORD;
	///Pin 1.21 - Latest measurement value for pin's input signal.
	AI_RAW_u16_Heater2Temperature_AI AT %IW2078: WORD := 0;
	///Pin 1.21 - Array of 50 latest conversion values for pin's input signal.
	AI_ARR_u16_Heater2Temperature_AI AT %IW3276: ARRAY [1..50] OF WORD;
	///Pin 1.21 - Latest measurement value for pin's pull-up voltage.
	AIPU_RAW_u16_Heater2Temperature_AI AT %IW2071: WORD := 0;
	///Pin 1.21 - Array of 50 latest conversion values for pin's pull-up voltage.
	AIPU_ARR_u16_Heater2Temperature_AI AT %IW2926: ARRAY [1..50] OF WORD;
	///Pin 2.6 - Unfiltered digital input status.
	DI_RAW_q_Battery1ChargeRq_DI AT %IX821.13: BOOL := FALSE;
	///Pin 2.7 - Unfiltered digital input status.
	DI_RAW_q_Battery1DiscahrgeRq_DI AT %IX831.13: BOOL := FALSE;
	///Pin 2.8 - Unfiltered digital input status.
	DI_RAW_q_Battery2ChargeRq_DI AT %IX841.13: BOOL := FALSE;
	///Pin 2.9 - Unfiltered digital input status.
	DI_RAW_q_Batter2DischargeRq_DI AT %IX851.13: BOOL := FALSE;
	///Pin 2.16 - Unfiltered digital input status.
	DI_RAW_q_ChargePlugLockStatus_DI AT %IX901.13: BOOL := FALSE;
	///Pin 2.23 - Latest measurement value for pin's input signal.
	AI_RAW_u16_HeaterDiagnose_AI AT %IW2059: WORD := 0;
	///Pin 2.23 - Array of 50 latest conversion values for pin's input signal.
	AI_ARR_u16_HeaterDiagnose_AI AT %IW2326: ARRAY [1..50] OF WORD;
	///Pin 2.23 - Latest measurement value for pin's pull-up voltage.
	AIPU_RAW_u16_HeaterDiagnose_AI AT %IW2073: WORD := 0;
	///Pin 2.23 - Array of 50 latest conversion values for pin's pull-up voltage.
	AIPU_ARR_u16_HeaterDiagnose_AI AT %IW3026: ARRAY [1..50] OF WORD;
	///Pin 3.5 - Unfiltered digital input status.
	DI_RAW_q_DirectionSwitch_ReverseCrawl_DI AT %IX980.8: BOOL := FALSE;
	///Pin 3.6 - Unfiltered digital input status.
	DI_RAW_q_DirectionSwitch_Drive_DI AT %IX990.8: BOOL := FALSE;
	///Pin 3.7 - Unfiltered digital input status.
	DI_RAW_q_IlluminiationStatsus_DI AT %IX881.13: BOOL := FALSE;
	///Pin 3.8 - Unfiltered digital input status.
	DI_RAW_q_DirectionSwitch_Reverse_DI AT %IX940.8: BOOL := FALSE;
	///Pin 3.9 - Unfiltered digital input status.
	DI_RAW_q_DirectionSwitch_DriveCrawl_DI AT %IX950.8: BOOL := FALSE;
	///Pin 3.11 - Unfiltered digital input status.
	DI_RAW_q_DirectionSwitch_Neutral_DI AT %IX960.8: BOOL := FALSE;
	///Pin 3.12 - Unfiltered digital input status.
	DI_RAW_q_DoorOpen_DI AT %IX970.8: BOOL := FALSE;
	///Pin 3.14 - Latest measurement value for pin's input signal.
	AI_RAW_u16_HeaterDiagnose2_AI AT %IW2079: WORD := 0;
	///Pin 3.14 - Array of 50 latest conversion values for pin's input signal.
	AI_ARR_u16_HeaterDiagnose2_AI AT %IW3326: ARRAY [1..50] OF WORD;
	///Pin 3.14 - Latest measurement value for pin's pull-up voltage.
	AIPU_RAW_u16_HeaterDiagnose2_AI AT %IW2075: WORD := 0;
	///Pin 3.14 - Array of 50 latest conversion values for pin's pull-up voltage.
	AIPU_ARR_u16_HeaterDiagnose2_AI AT %IW3126: ARRAY [1..50] OF WORD;
	///Pin 3.15 - Latest measurement value for pin's input signal.
	AI_RAW_u16_VehicleThrottlePedal1_AI AT %IW2060: WORD := 0;
	///Pin 3.15 - Array of 50 latest conversion values for pin's input signal.
	AI_ARR_u16_VehicleThrottlePedal1_AI AT %IW2376: ARRAY [1..50] OF WORD;
	///Pin 3.15 - Latest measurement value for pin's pull-up voltage.
	AIPU_RAW_u16_VehicleThrottlePedal1_AI AT %IW2083: WORD := 0;
	///Pin 3.15 - Array of 50 latest conversion values for pin's pull-up voltage.
	AIPU_ARR_u16_VehicleThrottlePedal1_AI AT %IW3526: ARRAY [1..50] OF WORD;
	///Pin 3.16 - Latest measurement value for pin's input signal.
	AI_RAW_u16_VehicleThrottlePedal2_AI AT %IW2080: WORD := 0;
	///Pin 3.16 - Array of 50 latest conversion values for pin's input signal.
	AI_ARR_u16_VehicleThrottlePedal2_AI AT %IW3376: ARRAY [1..50] OF WORD;
	///Pin 3.16 - Latest measurement value for pin's pull-up voltage.
	AIPU_RAW_u16_VehicleThrottlePedal2_AI AT %IW2085: WORD := 0;
	///Pin 3.16 - Array of 50 latest conversion values for pin's pull-up voltage.
	AIPU_ARR_u16_VehicleThrottlePedal2_AI AT %IW3626: ARRAY [1..50] OF WORD;
	///Pin 3.22 - Unfiltered digital input status.
	DI_RAW_q_VehicleKL15_DI AT %IX1010.8: BOOL := FALSE;
	///Pin 3.23 - Unfiltered digital input status.
	DI_RAW_q_VehicleKL51_DI AT %IX1020.8: BOOL := FALSE;
	///Pin 3.28 - Digital input state for pin.
	DI_RAW_q_HeaterIn_DI AT %IX768.4: BOOL := FALSE;
	///Pin 3.29 - Raw value for output pin Voltage measurement.
	AI_RAW_q_HeaterOut_DI AT %IW2082: WORD := 0;
	///Pin 3.29 - 50 latest conversion result for voltage measurement.
	AI_ARR_q_HeaterOut_DI AT %IW3476: ARRAY [1..50] OF WORD;
	///Pin 3.30 - Raw value for output pin Voltage measurement.
	AI_RAW_q_DrivetrainInverterRf1_DO AT %IW2088: WORD := 0;
	///Pin 3.30 - 50 latest conversion result for voltage measurement.
	AI_ARR_q_DrivetrainInverterRf1_DO AT %IW3776: ARRAY [1..50] OF WORD;
	///Pin 3.31 - Raw value for output pin Voltage measurement.
	AI_RAW_q_DrivetrainInverterRf2_DO AT %IW2086: WORD := 0;
	///Pin 3.31 - 50 latest conversion result for voltage measurement.
	AI_ARR_q_DrivetrainInverterRf2_DO AT %IW3676: ARRAY [1..50] OF WORD;
	///Pin 3.32 - Raw value for output pin Voltage measurement.
	AI_RAW_q_DrivetrainDCDCInhibit_DO AT %IW2092: WORD := 0;
	///Pin 3.32 - 50 latest conversion result for voltage measurement.
	AI_ARR_q_DrivetrainDCDCInhibit_DO AT %IW3976: ARRAY [1..50] OF WORD;
	///Pin 3.33 - Raw value for output pin Voltage measurement.
	AI_RAW_q_ChargePlugLED_Green_DO AT %IW2090: WORD := 0;
	///Pin 3.33 - 50 latest conversion result for voltage measurement.
	AI_ARR_q_ChargePlugLED_Green_DO AT %IW3876: ARRAY [1..50] OF WORD;
	///Pin 3.34 - Raw value for output pin Voltage measurement.
	AI_RAW_q_ChargePlugLED_Blue_DO AT %IW2063: WORD := 0;
	///Pin 3.34 - 50 latest conversion result for voltage measurement.
	AI_ARR_q_ChargePlugLED_Blue_DO AT %IW2526: ARRAY [1..50] OF WORD;
	///Pin 3.35 - Raw value for output pin Voltage measurement.
	AI_RAW_q_ChargePlugLED_Red_DO AT %IW2094: WORD := 0;
	///Pin 3.35 - 50 latest conversion result for voltage measurement.
	AI_ARR_q_ChargePlugLED_Red_DO AT %IW4076: ARRAY [1..50] OF WORD;
END_VAR

// Application/CodeTemplate/Globals/J1939Globals
VAR_GLOBAL
	J1939_CAN1: J1939_CAN1;
	J1939_FB_CAN1: J1939;
	J1939_CAN4: J1939_CAN4;
	J1939_FB_CAN4: J1939;
END_VAR

// Application/CodeTemplate/Globals/OD1_VAR
VAR_GLOBAL
	///Sub0: Information about the device type
	OD_DeviceType_Device1: UDINT := 405;
	///Sub0: Error information
	OD_ErrorReg_Device1: USINT := 0;
	///Sub1: Vendor ID
	///Sub2: Product code
	///Sub3: Revision number
	///Sub4: Serial number
	OD_IdentityArray_Device: ARRAY[1..4] OF UDINT;
	///Sub1: CodesysVersion
	OD_ToolsVersionInfo: ARRAY[1..1] OF DWORD := [50659328];
	///Sub0: TPDO Dummy Variable
	OD_CAN1_TPDO_DUMMY: BYTE := 0;
	///Sub0: RPDO Dummy Variable
	OD_CAN1_RPDO_DUMMY: BYTE := 0;
	///Sub1: Application version
	///Sub2: Additional version information
	///Sub3: Reserved for future use
	///Sub4: Reserved for future use
	///Sub5: Reserved for future use
	///Sub6: Reserved for future use
	///Sub7: Reserved for future use
	///Sub8: Reserved for future use
	///Sub9: Reserved for future use
	///Sub10: Reserved for future use
	OD_SoftwareInformation: ARRAY[1..10] OF STRING(79) := [''];
	///Sub1: MAC address byte 1
	///Sub2: MAC address byte 2
	///Sub3: MAC address byte 3
	///Sub4: MAC address byte 4
	///Sub5: MAC address byte 5
	///Sub6: MAC address byte 6
	OD_MACAddress: ARRAY[1..6] OF BYTE := [6(0)];
	///Sub1: Ethernet enabled/disabled
	///Sub2: DHCP on/off
	///Sub3: Reserved
	///Sub4: Reserved
	///Sub5: Reserved
	///Sub6: Reserved
	///Sub7: Reserved
	///Sub8: Reserved
	///Sub9: Reserved
	///Sub10: Reserved
	///Sub11: Reserved
	///Sub12: Reserved
	///Sub13: Reserved
	///Sub14: Reserved
	///Sub15: Reserved
	///Sub16: Reserved
	///Sub17: Reserved
	///Sub18: Netstatus
	///Sub19: IP address highest byte
	///Sub20: IP address 3rd byte
	///Sub21: IP address 2nd byte
	///Sub22: IP address lowest byte
	///Sub23: Gateway highest byte
	///Sub24: Gateway 3rd byte
	///Sub25: Gateway 2nd byte
	///Sub26: Gateway lowest byte
	///Sub27: Netmask highest byte
	///Sub28: Netmask 3rd byte
	///Sub29: Netmask 2nd byte
	///Sub30: Netmask first byte
	///Sub31: Reserved
	///Sub32: Reserved
	///Sub33: Reserved
	///Sub34: Reserved
	///Sub35: Reserved
	///Sub36: Reserved
	///Sub37: Reserved
	///Sub38: Reserved
	///Sub39: Reserved
	///Sub40: Reserved
	///Sub41: Reserved
	///Sub42: Reserved
	///Sub43: Reserved
	///Sub44: Reserved
	///Sub45: Reserved
	///Sub46: Reserved
	///Sub47: Reserved
	///Sub48: Reserved
	///Sub49: Reserved
	///Sub50: Reserved
	OD_EthernetConfiguration: ARRAY[1..50] OF BYTE := [50(0)];
	///Sub1: CODESYS communication enabled
	///Sub2: CODESYS communication node-ID
	///Sub3: Bit rate
	///Sub4: Cable detection offset for CODESYS node-ID
	///Sub5: Cable detection offset for PLCopen node-ID
	///Sub6: Mask for cable detection pins
	///Sub7: Reserved
	///Sub8: Reserved
	///Sub9: Reserved
	///Sub10: PLCopen application node-ID in CAN1
	OD_G_CAN1_Comms: ARRAY[1..10] OF WORD := [10(0)];
	///Sub1: CODESYS communication enabled
	///Sub2: CODESYS communication node-ID
	///Sub3: Bit rate
	///Sub4: Reserved
	///Sub5: Reserved
	///Sub6: Reserved
	///Sub7: Reserved
	///Sub8: Reserved
	///Sub9: Reserved
	///Sub10: PLCopen application node-ID in CAN2
	OD_G_CAN2_Comms: ARRAY[1..10] OF WORD := [10(0)];
	///Sub1: CODESYS communication enabled
	///Sub2: CODESYS communication node-ID
	///Sub3: Bit rate
	///Sub4: Reserved
	///Sub5: Reserved
	///Sub6: Reserved
	///Sub7: Reserved
	///Sub8: Reserved
	///Sub9: Reserved
	///Sub10: PLCopen application node-ID in CAN3
	OD_G_CAN3_Comms: ARRAY[1..10] OF WORD := [10(0)];
	///Sub1: CODESYS communication enabled
	///Sub2: CODESYS communication node-ID
	///Sub3: Bit rate
	///Sub4: Reserved
	///Sub5: Reserved
	///Sub6: Reserved
	///Sub7: Reserved
	///Sub8: Reserved
	///Sub9: Reserved
	///Sub10: PLCopen application node-ID in CAN4
	OD_G_CAN4_Comms: ARRAY[1..10] OF WORD := [10(0)];
	/// 16#2131 Parameter CSV unique ID
	OD_Parameter_CSV_unique_ID1: UINT := 16#0000;
END_VAR

// Application/CodeTemplate/Globals/OD2_VAR
VAR_GLOBAL
	///Sub0: Information about the device type
	OD_DeviceType_Device2: UDINT := 405;
	///Sub0: Error information
	OD_ErrorReg_Device2: USINT := 0;
	///Sub0: TPDO Dummy Variable
	OD_CAN2_TPDO_DUMMY: BYTE := 0;
	///Sub0: RPDO Dummy Variable
	OD_CAN2_RPDO_DUMMY: BYTE := 0;
	/// 16#2131 Parameter CSV unique ID
	OD_Parameter_CSV_unique_ID2: UINT := 16#0000;
END_VAR

// Application/CodeTemplate/Globals/OD3_VAR
VAR_GLOBAL
	///Sub0: Information about the device type
	OD_DeviceType_Device3: UDINT := 405;
	///Sub0: Error information
	OD_ErrorReg_Device3: USINT := 0;
	///Sub0: PDO Dummy Variable
	OD_CAN3_PDO_DUMMY: BYTE := 0;
	/// 16#2131 Parameter CSV unique ID
	OD_Parameter_CSV_unique_ID3: UINT := 16#0000;
END_VAR

// Application/CodeTemplate/Globals/OD4_VAR
VAR_GLOBAL
	///Sub0: Information about the device type
	OD_DeviceType_Device4: UDINT := 405;
	///Sub0: Error information
	OD_ErrorReg_Device4: USINT := 0;
	///Sub0: PDO Dummy Variable
	OD_CAN4_PDO_DUMMY: BYTE := 0;
	/// 16#2131 Parameter CSV unique ID
	OD_Parameter_CSV_unique_ID4: UINT := 16#0000;
END_VAR

// Application/CodeTemplate/Globals/Slave_Configurations
VAR_GLOBAL
END_VAR

// Application/CodeTemplate/Globals/SYSTEM
VAR_GLOBAL
	SYSTEM_ProjectInfo: APPLICATION_INFO;
	SYSTEM_FW_VERSION: STRING(79) := 'X.X.X';
	///Type for control unit.
	SYSTEM_ControlUnitType: DWORD := 0;
	///Revision for control unit
	SYSTEM_ControlUnitRevision: DWORD := 0;
	///Serial number for control unit
	SYSTEM_SerialNumber: DWORD := 0;
	///Vendor-ID which is read from firmware
	SYSTEM_VendorId: DWORD := 0;
	///Pointer to 5050 FW side error log. This is read-only area, all writings will cause access error.
	SYSTEM_FW_Error_Log: POINTER TO SysErrorLogData;
END_VAR

// Application/UserCode/BMS/BMS_VAR
VAR_GLOBAL
	(*BMS data taken from each BMS type to be used by the main program*)
	gu8_BMS_SOC						:	USINT;
	gr_BMS_BatteryVoltage			:	REAL;
	gs16_BMS_BatteryCurrent			:	INT;
	gu16_BMS_AverageCellVoltage		:	UINT;
	gu16_BMS_LowCellVoltage			:	UINT;
	gu16_BMS_HighCellVoltage		:	UINT;
	gr_BMS_AverageTemp				:	REAL;
	gr_BMS_LowTemp					:	REAL;
	gr_BMS_HighTemp					:	REAL;
	gr_BMS_DCL						:	REAL;
	gr_BMS_CCL						:	REAL;
	gu16_BMS_MinimumPackVoltage		:	UINT;
	gu16_BMS_Maximum_Pack_Voltage	:	UINT;
	gr_BMS1_Voltage					:	REAL;
	gr_BMS2_Voltage					:	REAL;
	gs16_BMS1_CCL					:	INT;
	gs16_BMS2_CCL					:	INT;
	gu16_BMS1_LowCellVoltage		:	UINT;
	gu16_BMS2_LowCellVoltage		:	UINT;
	gu16_BMS1_HighCellVoltage		:	UINT;
	gu16_BMS2_HighCellVoltage		:	UINT;
	gu16_BMS1_LowCellVoltage_ID		:	UINT;
	gu16_BMS2_LowCellVoltage_ID		:	UINT;
	gu16_BMS1_HighCellVoltage_ID	:	UINT;
	gu16_BMS2_HighCellVoltage_ID	:	UINT;
END_VAR

VAR_GLOBAL CONSTANT
	CONTACTORSWITCH_CURRENT_LIMIT	:	USINT	:=	3; (*Assigned an intial value of 10A*)
END_VAR

// Application/UserCode/BMS/BMS_VAR_1
VAR_GLOBAL
	(*BMS data taken from each BMS type to be used by the main program*)
	gu8_BMS_SOC						:	USINT;
	gr_BMS_BatteryVoltage			:	REAL;
	gs16_BMS_BatteryCurrent			:	INT;
	gu16_BMS_AverageCellVoltage		:	UINT;
	gu16_BMS_LowCellVoltage			:	UINT;
	gu16_BMS_HighCellVoltage		:	UINT;
	gr_BMS_AverageTemp				:	REAL;
	gr_BMS_LowTemp					:	REAL;
	gr_BMS_HighTemp					:	REAL;
	gr_BMS_DCL						:	REAL;
	gr_BMS_CCL						:	REAL;
	gu16_BMS_MinimumPackVoltage		:	UINT;
	gu16_BMS_Maximum_Pack_Voltage	:	UINT;
	gr_BMS1_Voltage					:	REAL;
	gr_BMS2_Voltage					:	REAL;
	gs16_BMS1_CCL					:	INT;
	gs16_BMS2_CCL					:	INT;
	gu16_BMS1_LowCellVoltage		:	UINT;
	gu16_BMS2_LowCellVoltage		:	UINT;
	gu16_BMS1_HighCellVoltage		:	UINT;
	gu16_BMS2_HighCellVoltage		:	UINT;
	gu16_BMS1_LowCellVoltage_ID		:	UINT;
	gu16_BMS2_LowCellVoltage_ID		:	UINT;
	gu16_BMS1_HighCellVoltage_ID	:	UINT;
	gu16_BMS2_HighCellVoltage_ID	:	UINT;
END_VAR

// Application/UserCode/CAN1/CAN1_VAR_1
VAR_GLOBAL
	(*Tx variables*)
	(*EEC1*)
	gu8_ENG_EngineTorqueMode					:	USINT;
	gu8_ENG_ActlEngPrcntTorqueHghResolution_Tx	:	USINT;
	gu8_ENG_DriversDemandEnginePercentTorque	:	USINT;
	gu8_ENG_ActualEnginePercentTorque			:	USINT;
	gu16_ENG_EngineSpeed_Tx						:	UINT;
	gu8_ENG_SrcAddrOfCtrllingDevForEngCtrl		:	USINT;
	gu8_ENG_EngineStarterMode					:	USINT;
	gu8_ENG_EngineDemandPercentTorque			:	USINT;
	(*EEC2*)
	gu8_ENG_AccelPedal1LowIdleSwitch			:	USINT;
	gu8_ENG_AccelPedalKickdownSwitch			:	USINT;
	gu8_ENG_RoadSpeedLimitStatus				:	USINT;
	gu8_ENG_AccelPedal2LowIdleSwitch			:	USINT;
	gu8_ENG_AccelPedalPosition_Tx				:	USINT;
	gu8_ENG_EnginePercLoadCurrentSpeed			:	USINT;
	gu8_ENG_RemoteAccelPedalPosition_Tx			:	USINT;
	gu8_ENG_AccelPedalPosition2_Tx				:	USINT;
	gu8_ENG_VehicleAccelRateLimitStatus			:	USINT;
	gu8_ENG_MomentaryEngMaxPowEnableFeedback	:	USINT;
	gu8_ENG_DPFThermalManagementActive			:	USINT;
	gu8_ENG_SCRThermalManagementActive			:	USINT;
	gu8_ENG_ActualMaxAvailableEngPercTorque_Tx	:	USINT;
	gu8_ENG_EstimatedPumpingPercentTorque		:	USINT;
	(*EEC3*)
	gu8_ENG_NominalFrictionPercTorque				:	USINT;
	gu16_ENG_EngDesiredOperatingSpeed_Tx			:	UINT;
	gu8_ENG_EngDesiredOperatingSpeedAsymAdjust		:	USINT;
	gu8_ENG_EstEngParasiticLossPercTorque			:	USINT;
	gu16_ENG_Aftertreatment1ExhaustGasMassFlow_Tx	:	UINT;
	gu8_ENG_Aftertreatment1IntakeDewPoint			:	USINT;
	gu8_ENG_Aftertreatment1ExhaustDewPoint			:	USINT;
	gu8_ENG_Aftertreatment2IntakeDewPoint			:	USINT;
	gu8_ENG_Aftertreatment2ExhaustDewPoint			:	USINT;
	(*CCSS*)
	gu8_ENG_MaxVehicleSpeedLimit				:	USINT;
	gu8_ENG_CruiseControlHighSetSpeedLimit		:	USINT;
	gu8_ENG_CruiseControlLowSetSpeedLimit		:	USINT;
	
	(*Tx preconversion*)
	(*EEC1*)
	gr_ENG_ActlEngPrcntTorqueHghResolution		:	REAL;
	gr_ENG_EngineSpeed							:	REAL;
	(*EEC2*)
	gr_ENG_AccelPedalPosition1					:	REAL;
	gr_ENG_RemoteAccelPedalPosition				:	REAL;
	gr_ENG_AccelPedalPosition2					:	REAL;
	gr_ENG_ActualMaxAvailableEngPercTorque		:	REAL;
	(*EEC3*)
	gr_ENG_EngDesiredOperatingSpeed				:	REAL;
	gr_ENG_AfterTreatment1ExhaustGasMassFlow	:	REAL;
	
	
	(*Rx Variables*)
	gq_Dennis_Accel_NewData						:	BOOL;
	gu8_AccelPedal_Dennis_Rx					:	USINT;
	gq_BrakePedal_Dennis_Rx						:	BOOL;
	gu8_BrakePedal_Perc_Dennis_Rx				:	USINT;
	gu8_GearSelector_Dennis_Rx					:	USINT;
	gq_Neutral_Dennis_Rq						:	BOOL;
	gq_Drive_Dennis_Rq							:	BOOL;
	gq_Reverse_Dennis_Rq						:	BOOL;
	
	gu8_Dennis_AirPressureSusp_Rx				:	USINT;
	gu8_Dennis_AirPressureBrake1_Rx				:	USINT;
	gu8_Dennis_AirPressureBrake2_Rx				:	USINT;
	
	(*EBC1*)
	gu8_EBC1_ASREngineControlActive				:	USINT;
	gu8_EBC1_ASRBrakeControlActive				:	USINT;
	gu8_EBC1_ABSActive							:	USINT;
	gu8_EBC1_EBSBrakeSwitch						:	USINT;
	gu8_EBC1_BrakePedalPosition					:	USINT;
	gu8_EBC1_ABSOffroadSwitch					:	USINT;
	gu8_EBC1_ASROffroadSwitch					:	USINT;
	gu8_EBC1_ASRHillholderSwitch				:	USINT;
	gu8_EBC1_TractionControlOverrideSwtich		:	USINT;
	gu8_EBC1_AcceleratorInterlockSwitch			:	USINT;
	gu8_EBC1_EngineDerateSwitch					:	USINT;
	gu8_EBC1_EngineAuxiliaryShutdownSwitch		:	USINT;
	gu8_EBC1_RemoteAcceleratorEnableSwitch		:	USINT;
	gu8_EBC1_EngineRetarderSelection			:	USINT;
	gu8_EBC1_ABSFullyOperational				:	USINT;
	gu8_EBC1_gu8_EBC1_EBSRedWarningSignal		:	USINT;
	gu8_EBC1_ABSEBSAmberWarningSignal			:	USINT;
	gu8_EBC1_ATCASRInformationSignal			:	USINT;
	gu8_EBC1_SrcAddrOfCrtllingDevForBrkCtrl		:	USINT;
	gu8_EBC1_HaltBrakeSwitch					:	USINT;
	gu8_EBC1_TrailerABSStatus					:	USINT;
	gu8_EBC1_TractorMntdTrailerABSWarningSignal	:	USINT;
	
	(*EBC2*)
	gu16_EBC2_KB_FrontAxleSpeed_Rx				:	UINT;
	gu16_EBC2_KB_FrontLeftRelSpd_Rx				:	USINT;
	gu16_EBC2_KB_FrontRightRelSpd_Rx			:	USINT;
	gu16_EBC2_KB_RearLeft1RelSpd_Rx				:	USINT;
	gu16_EBC2_KB_RearRight1RelSpd_Rx			:	USINT;
	gu16_EBC2_KB_RearLeft2RelSpd_Rx				:	USINT;
	gu16_EBC2_KB_RearRight2RelSpd_Rx			:	USINT;
	
	gr_EBC2_KB_FrontAxleSpeed				:	REAL;
	gr_EBC2_KB_FrontLeftRelSpd				:	REAL;
	gr_EBC2_KB_FrontRightRelSpd				:	REAL;
	gr_EBC2_KB_RearLeft1RelSpd				:	REAL;
	gr_EBC2_KB_RearRight1RelSpd				:	REAL;
	gr_EBC2_KB_RearLeft2RelSpd				:	REAL;
	gr_EBC2_KB_RearRight2RelSpd				:	REAL;
	
	gu8_RegenStick01Pos						:	USINT;
	gu8_RegenStick12Pos						:	USINT;
	
	(*Dennis CAN1 Comms loss*)
	gq_Dennis_CAN1_CommsLoss					:	BOOL;
	
	gq_ABSActive								:	BOOL;
	
	(*Allison*)
	gu8_ETC7_TransmissionEngaged_Tx				:	USINT;
	gu8_ProbA_GearSelected_Tx					:	USINT;

	
	gq_Bob_Handbrake_CAN	:	BOOL;
	gq_Bob_Brake_CAN		:	BOOL;
	gu8_Bob_BrakePos_CAN	:	USINT;
	
	gu8_Bob_Accel_CAN		:	USINT;
	gr_Bob_Accel			:	REAL;
	gu8_Bob_RegenSelector_CAN	:	USINT;
	
	gu16_Bob_RightDrive_CAN	:	UINT;
	gu16_Bob_LeftDrive_CAN	:	UINT;
	gu16_Bob_RightFront_CAN	:	UINT;
	gu16_Bob_LeftFront_CAN	:	UINT;
	
	gu8_Bob_ServiceBrakeAirPressCircuit1_CAN	:	USINT;
	gu8_Bob_ServiceBrakeAirPressCircuit2_CAN	:	USINT;
	gu8_Bob_AirSuspensionSupplyPress_CAN		:	USINT;
	
	gr_Bob_ServiceBrakeAirPressCircuit1		:	REAL;
	gr_Bob_ServiceBrakeAirPressCircuit2		:	REAL;
	gr_Bob_AirSuspensionSupplyPress			:	REAL;
	
	gu8_Merc_AirComepressor_Rq	:	USINT;
	gq_Merc_AirComp_Rq		:	BOOL;
	gq_Merc_AirComp_Enabled	:	BOOL;
	
	gu16_RPM_Display	:	UINT;
	gq_StabTracDisable_Rx	:	BOOL;
	gq_Bob_WheelSpeedSensor_Fail	:	BOOL;
	
	gu16_MCM02_EngineTorque_Tx	:	UINT;
	gu16_TCM03_ShaftSpeed_Tx	:	UINT;
	
END_VAR

// Application/UserCode/CAN3/CAN3_VAR_1
VAR_GLOBAL
	
	gu8_GearSelector_Bob_Rx	:	USINT	:=	0;
	gq_Neutral_Bob_Rq	:	BOOL;
	gq_Drive_Bob_Rq		:	BOOL;
	gq_Reverse_Bob_Rq	:	BOOL;
	
	gu8_Merc_AutoManualSwitch	:	USINT;
	gu8_Merc_GearSelectSwitch	:	USINT;
	gq_Merc_Neutral				:	BOOL;
	gq_Merc_Drive				:	BOOL;
	gq_Merc_Reverse				:	BOOL;
END_VAR

// Application/UserCode/CAN4/CAN4_VAR
VAR_GLOBAL
	gu16_CurrentGear	:	UINT;
	gu16_CurrentGear1	:	UINT;
	gu8_CurrentGear2	:	USINT;
	
	gq_Handbrake_CAN	:	BOOL;
	
	(*********************************************)
	(*601*)
	gu16_CAN4_TripCounter_km_Tx			:	UINT;
	gu16_CAN4_DisplayRangeMin_Tx		:	UINT;
	gu16_CAN4_DisplayRangeMax_Tx		:	UINT;
	gu16_CAN4_DisplayRangeEst_Tx		:	UINT;
	(*201*)
	gs8_CAN4_CruiseControlSetpoint_Tx	:	SINT;
	gs8_CAN4_DummyScreen601_Tx			:	SINT;
	gs8_CAN4_DisplayTemp_Tx				:	SINT;
	gs8_CAN4_DisplayDirection_Tx		:	SINT;
	gs8_CAN4_SOC_Tx						:	SINT;
	gs8_CAN4_DispVehicleStatus_Tx		:	SINT;
	gs8_CAN4_PowerIndicationRelative_Tx	:	SINT;
	gs8_CAN4_DisplayStatus_Tx			:	SINT;
	(*301*)
	gs8_CAN4_SOC1_Tx					:	SINT;
	gs8_CAN4_BatteryVoltage_Tx			:	SINT;
	gs8_CAN4_MotorTemp_Tx				:	SINT;
	gs8_CAN4_InverterTemp_Tx			:	SINT;
	gu8_CAN4_ChargerStatus_Tx			:	USINT;
	gq_CAN4_ChargerPP_Tx				:	BOOL;
	gs8_CAN4_ThrottlePedal_Tx			:	SINT;
	gs8_CAN4_BrakePedal_Tx				:	SINT;
	gs8_CAN4_VehicleSpeedMsg_Tx			:	SINT;
	(*401*)
	gs8_CAN4_VehicleStatus_Tx			:	SINT;
	gs8_CAN4_RegenTorquePercDisplay_Tx	:	SINT;
	gs16_CAN4_PowerIndication_Tx		:	INT;
	gs16_CAN4_BatteryCurrent_Tx			:	INT;
	
	(*********************************************)
	(**)
	gq_Dash_Sevcon1_Enable	:	BOOL;
	gq_Dash_Sevcon2_Enable	:	BOOL;
	gq_Dash_Charge_Rq		:	BOOL;
	gq_Dash_Discharge_Rq	:	BOOL;
	gs16_Dash_BattCurrent_Tx	:	INT;
	gu8_Dash_AccelPedal_Tx	:	USINT;
	gu8_Dash_BrakePressure1_Tx	:	USINT;
	gu8_Dash_BrakePressure2_Tx	:	USINT;
	gq_BattFullyCharged	:	BOOL;
	gs16_Dash_Power	:	INT;
	gs8_Dash_AverageTemp_Tx	:	SINT;
	gs8_Dash_HighTemp_Tx	:	SINT;
	gs8_Dash_LowTemp_Tx	:	SINT;
	
	gu8_BMS1_LowCellV_Tx	:	USINT;
	gu8_BMS2_LowCellV_Tx	:	USINT;
	
	gu16_TCM2_OutputShaftSpeed	:	UINT;
	gu8_TCM2_DrvDirec_Stat		:	USINT;
	gu8_TCM2_RotSens_Stat		:	USINT;
	gu8_TCM8_Gear				:	USINT;
	gu8_TCM8_DrvDirByGr_Stat	:	USINT;
	gu16_TCM11_ActualGearRatio	:	UINT;
	gu8_Compressor_Temp_To_Screen: BYTE;
END_VAR

// Application/UserCode/CAN4/HMI_VAR
VAR_GLOBAL
	(* COBID	:=	16#57B, *)
	
	qq_Spare_0_0			:BOOL;
	qq_Spare_0_1			:BOOL;	
	gq_HMI_Heater_Enable	:BOOL := FALSE;
	qq_Spare_0_3			:BOOL;
	qq_Spare_0_4			:BOOL;
	gq_HMI_Heater_Low		:BOOL;
	gq_HMI_Heater_Med		:BOOL;
	gq_HMI_Heater_Hi		:BOOL;
	
	qq_BMS1_PB_DTC_Reset	:BOOL;
	qq_BMS2_PB_DTC_Reset	:BOOL;
	qq_Spare_1_2			:BOOL;
	qq_Spare_1_3			:BOOL;
	qq_Spare_1_4			:BOOL;
	qq_Spare_1_5			:BOOL;
	qq_Spare_1_6			:BOOL;
	qq_Spare_1_7			:BOOL;
	
	qu8_HMI_Spare_2			:BYTE;
	qu8_HMI_Spare_3			:BYTE;
	qu8_HMI_Spare_4			:BYTE;
	qu8_HMI_Spare_5			:BYTE;
	qu8_HMI_Spare_6			:BYTE;
	qu8_HMI_Spare_7			:BYTE;
END_VAR

// Application/UserCode/CAN4/CAN4_VAR_1
VAR_GLOBAL
	gu16_CurrentGear	:	UINT;
	gu16_CurrentGear1	:	UINT;
	gu8_CurrentGear2	:	USINT;
	
	gq_Handbrake_CAN	:	BOOL;
	
	(*********************************************)
	(*601*)
	gq_Dash_Sevcon1_Enable	:	BOOL;
	gq_Dash_Sevcon2_Enable	:	BOOL;
	gq_Dash_Charge_Rq		:	BOOL;
	gq_Dash_Discharge_Rq	:	BOOL;
	gs16_Dash_BattCurrent_Tx	:	INT;
	gu8_Dash_AccelPedal_Tx	:	USINT;
	gu8_Dash_BrakePressure1_Tx	:	USINT;
	gu8_Dash_BrakePressure2_Tx	:	USINT;
	gq_BattFullyCharged	:	BOOL;
	gs16_Dash_Power	:	INT;
	
	gu16_TCM2_OutputShaftSpeed	:	UINT;
	gu8_TCM2_DrvDirec_Stat		:	USINT;
	gu8_TCM2_RotSens_Stat		:	USINT;
	gu8_TCM8_Gear				:	USINT;
	gu8_TCM8_DrvDirByGr_Stat	:	USINT;
	gu16_TCM11_ActualGearRatio	:	UINT;
END_VAR

// Application/UserCode/ePTO/ePTO_VAR
VAR_GLOBAL
	gu8_ePTO_ActivationByte	:	USINT;
	gq_ePTO_Activate		:	BOOL;
	gs16_InverterTemp		:	INT;
	gs16_MotorTemp			:	INT;
	gu16_TrqHi				:	UINT;
	gu16_TrqLo				:	UINT;
	gu8_Asym_Limits			:	USINT;
	gu8_DIGITAL1			: USINT	:=	16#0;
	gu16_Skai_SpeedTarget	:	UINT;
	
	gu8_CANOpen_Command		:	USINT;
	gu8_CANOpen_NodeAddress	:	USINT;
	
	gq_ePTO_FanEnable		:	BOOL;
END_VAR

// Application/UserCode/ePTO/ePTO_VAR_1
VAR_GLOBAL
	gu8_ePTO_ActivationByte	:	USINT;
	gq_ePTO_Activate		:	BOOL;
	gs16_InverterTemp		:	INT;
	gs16_MotorTemp			:	INT;
	gu16_TrqHi				:	UINT;
	gu16_TrqLo				:	UINT;
	gu8_Asym_Limits			:	USINT;
	gu8_DIGITAL1			: USINT	:=	16#0;
	gu16_Skai_SpeedTarget	:	UINT;
	
	gu8_CANOpen_Command		:	USINT;
	gu8_CANOpen_NodeAddress	:	USINT;
	
END_VAR

// Application/UserCode/Fault Handler/Fault_VAR
VAR_GLOBAL
	gq_BMS1_Orion_Error			:	BOOL;
	gq_BMS2_Orion_Error			:	BOOL;
	gq_BMS1_Error				:	BOOL;
	gq_BMS2_Error				:	BOOL;
	gq_BMS_Error				:	BOOL;
	gq_DCDC_Bel_Error			:	BOOL;
	gq_MCU_Error				:	BOOL;
	gq_NLG1_Error				:	BOOL;
	gq_NLG2_Error				:	BOOL;
	gq_Sevcon_Steer_Error		:	BOOL;
	gq_Sevcon_Compressor_Error	:	BOOL;
	gq_LV_Error					:	BOOL;
	
	gq_MCU_CutOff_LowCellV			:	BOOL;
	gq_DriveMode_CutOff_LowCellV	:	BOOL;
	
END_VAR

// Application/UserCode/Main Program/PersistentVars
VAR_GLOBAL PERSISTENT RETAIN
	gu8_BMSType: USINT := 1;
	gu8_ChassisType	:	USINT	:=	1;
	gu8_ChargerType	:	USINT	:=	1;
	gu16_CAN1_BaudRate	:	UINT	:=	250;
	gu16_CAN2_BaudRate	:	UINT	:=	500;
	gu16_CAN3_BaudRate	:	UINT	:=	500;
	gu16_CAN4_BaudRate	:	UINT	:=	250;
	SpeedOTG: REAL := 55;
	SpeedOTG1: REAL := 40;
	
	gu16_GearRatio_PreCF		:	UINT	:=	1000;
	gu16_DyfRatio_PreCF			:	UINT	:=	6428;
	gu16_TireWidth_mm			:	UINT	:=	315;
	gu8_TireProfile_Perc		:	USINT	:=	80;
	gu16_WheelDiameter_PreCF	:	UINT	:=	225;
	
	gr_VehicleAllTimeDistance			:	REAL;
	gq_Frosty_NoWheelSpeedSensors		:	BOOL	:=	FALSE;
	gq_BodyStepInstalled				:	BOOL	:=	FALSE;
	
	gq_Daimler_PowerShift_Installed		:	BOOL	:=	FALSE; (*Variable for if the system uses the chassis request for gear change or the Allison gearbox*)
	gq_APU_Installed					:	BOOL	:=	FALSE;
	gq_CAN1_Merc_Gears: BOOL := FALSE;
	E_Stop_Installed: BOOL := TRUE;
	// Sends all the messages the PS does but from pad control
	gq_Allison_Pad_Override: BOOL := FALSE;
	
END_VAR

